LIN {X 0,Y 617.563,Z 761.616,A -85,B 0,C 180,E1 7757.121,E2 7757.121} C_VEL
LIN {X 0,Y 618.923,Z 727.183,A -85,B 0,C 180,E1 7758.711,E2 7758.711} C_VEL
LIN {X 0,Y 620.162,Z 689.828,A -85,B 0,C 180,E1 7759.795,E2 7759.795} C_VEL
LIN {X 0,Y 620.989,Z 629.444,A -85,B 0,C 180,E1 7760.813,E2 7760.813} C_VEL
LIN {X 0,Y 611.333,Z 601.31,A -85,B 0,C 180,E1 7761.822,E2 7761.822} C_VEL
LIN {X 0,Y 611.227,Z 601.31,A -85,B 0,C 180,E1 7766.829,E2 7766.829} C_VEL
LIN {X 0,Y 611.22,Z 601.31,A -85,B 0,C 180,E1 7772.565,E2 7772.565} C_VEL
LIN {X 0,Y 611.08,Z 601.31,A -85,B 0,C 180,E1 7775.407,E2 7775.407} C_VEL
LIN {X 0,Y 607.041,Z 601.31,A -85,B 0,C 180,E1 7777.008,E2 7777.008} C_VEL
LIN {X 0,Y 603.157,Z 601.31,A -85,B 0,C 180,E1 7778.63,E2 7778.63} C_VEL
LIN {X 0,Y 603.164,Z 601.31,A -85,B 0,C 180,E1 7783.244,E2 7783.244} C_VEL
LIN {X 0,Y 603.063,Z 601.31,A -85,B 0,C 180,E1 7789.218,E2 7789.218} C_VEL
LIN {X 0,Y 603.149,Z 601.313,A -85,B 0,C 180,E1 7792.763,E2 7792.763} C_VEL
LIN {X 0,Y 619.848,Z 644.804,A -85,B 0,C 180,E1 7794.111,E2 7794.111} C_VEL
LIN {X 0,Y 624.51,Z 654.896,A -85,B 0,C 180,E1 7794.435,E2 7794.435} C_VEL
LIN {X 0,Y 623.787,Z 712.423,A -85,B 0,C 180,E1 7795.241,E2 7795.241} C_VEL
LIN {X 0,Y 621.771,Z 758.458,A -85,B 0,C 180,E1 7796.44,E2 7796.44} C_VEL
LIN {X 0,Y 619.212,Z 802.863,A -85,B 0,C 180,E1 7798.211,E2 7798.211} C_VEL
LIN {X 0,Y 616.234,Z 843.726,A -85,B 0,C 180,E1 7800.453,E2 7800.453} C_VEL
LIN {X 0,Y 613.148,Z 881.254,A -85,B 0,C 180,E1 7803.152,E2 7803.152} C_VEL
LIN {X 0,Y 610.305,Z 914.42,A -85,B 0,C 180,E1 7806.211,E2 7806.211} C_VEL
LIN {X 0,Y 607.707,Z 941.239,A -85,B 0,C 180,E1 7809.574,E2 7809.574} C_VEL
LIN {X 0,Y 605.902,Z 964.248,A -85,B 0,C 180,E1 7813.291,E2 7813.291} C_VEL
LIN {X 0,Y 604.836,Z 983.335,A -85,B 0,C 180,E1 7817.388,E2 7817.388} C_VEL
LIN {X 0,Y 604.309,Z 996.172,A -85,B 0,C 180,E1 7821.352,E2 7821.352} C_VEL
LIN {X 0,Y 604.218,Z 1003.674,A -85,B 0,C 180,E1 7824.969,E2 7824.969} C_VEL
LIN {X 0,Y 604.188,Z 1007.166,A -85,B 0,C 180,E1 7828.567,E2 7828.567} C_VEL
LIN {X 0,Y 604.173,Z 1006.211,A -85,B 0,C 180,E1 7832.879,E2 7832.879} C_VEL
LIN {X 0,Y 604.211,Z 1001.191,A -85,B 0,C 180,E1 7836.484,E2 7836.484} C_VEL
LIN {X 0,Y 604.502,Z 989.708,A -85,B 0,C 180,E1 7840.84,E2 7840.84} C_VEL
LIN {X 0,Y 605.347,Z 973.833,A -85,B 0,C 180,E1 7844.802,E2 7844.802} C_VEL
LIN {X 0,Y 606.845,Z 952.245,A -85,B 0,C 180,E1 7848.771,E2 7848.771} C_VEL
LIN {X 0,Y 609.432,Z 923.908,A -85,B 0,C 180,E1 7852.71,E2 7852.71} C_VEL
LIN {X 0,Y 612.346,Z 892.188,A -85,B 0,C 180,E1 7855.969,E2 7855.969} C_VEL
LIN {X 0,Y 615.619,Z 855.246,A -85,B 0,C 180,E1 7858.921,E2 7858.921} C_VEL
LIN {X 0,Y 618.871,Z 817.185,A -85,B 0,C 180,E1 7861.277,E2 7861.277} C_VEL
LIN {X 0,Y 622.102,Z 775.086,A -85,B 0,C 180,E1 7863.235,E2 7863.235} C_VEL
LIN {X 0,Y 624.782,Z 729.282,A -85,B 0,C 180,E1 7864.714,E2 7864.714} C_VEL
LIN {X 0,Y 626.356,Z 682.545,A -85,B 0,C 180,E1 7865.608,E2 7865.608} C_VEL
LIN {X 0,Y 626.28,Z 652.86,A -85,B 0,C 180,E1 7866.017,E2 7866.017} C_VEL
LIN {X 0,Y 603.192,Z 601.31,A -85,B 0,C 180,E1 7868.12,E2 7868.12} C_VEL
LIN {X 0,Y 603.121,Z 601.31,A -85,B 0,C 180,E1 7873.245,E2 7873.245} C_VEL
LIN {X 0,Y 603.083,Z 601.31,A -85,B 0,C 180,E1 7879.222,E2 7879.222} C_VEL
LIN {X 0,Y 603.121,Z 601.31,A -85,B 0,C 180,E1 7884.709,E2 7884.709} C_VEL
LIN {X 0,Y 603.248,Z 601.31,A -85,B 0,C 180,E1 7889.85,E2 7889.85} C_VEL
LIN {X 0,Y 603.366,Z 601.31,A -85,B 0,C 180,E1 7894.732,E2 7894.732} C_VEL
LIN {X 0,Y 603.462,Z 601.31,A -85,B 0,C 180,E1 7899.422,E2 7899.422} C_VEL
LIN {X 0,Y 603.517,Z 601.31,A -85,B 0,C 180,E1 7903.97,E2 7903.97} C_VEL
LIN {X 0,Y 603.64,Z 601.31,A -85,B 0,C 180,E1 7909.88,E2 7909.88} C_VEL
LIN {X 0,Y 603.837,Z 601.31,A -85,B 0,C 180,E1 7914.239,E2 7914.239} C_VEL
LIN {X 0,Y 603.903,Z 601.31,A -85,B 0,C 180,E1 7918.561,E2 7918.561} C_VEL
LIN {X 0,Y 603.929,Z 601.31,A -85,B 0,C 180,E1 7922.874,E2 7922.874} C_VEL
LIN {X 0,Y 603.718,Z 601.31,A -85,B 0,C 180,E1 7927.206,E2 7927.206} C_VEL
LIN {X 0,Y 603.614,Z 601.31,A -85,B 0,C 180,E1 7933.052,E2 7933.052} C_VEL
LIN {X 0,Y 603.565,Z 601.31,A -85,B 0,C 180,E1 7937.527,E2 7937.527} C_VEL
LIN {X 0,Y 603.457,Z 601.31,A -85,B 0,C 180,E1 7942.118,E2 7942.118} C_VEL
LIN {X 0,Y 603.371,Z 601.31,A -85,B 0,C 180,E1 7946.865,E2 7946.865} C_VEL
LIN {X 0,Y 603.25,Z 601.31,A -85,B 0,C 180,E1 7951.825,E2 7951.825} C_VEL
LIN {X 0,Y 603.163,Z 601.31,A -85,B 0,C 180,E1 7957.067,E2 7957.067} C_VEL
LIN {X 0,Y 603.143,Z 601.31,A -85,B 0,C 180,E1 7962.696,E2 7962.696} C_VEL
LIN {X 0,Y 603.084,Z 601.31,A -85,B 0,C 180,E1 7967.279,E2 7967.279} C_VEL
LIN {X 0,Y 603.101,Z 601.31,A -85,B 0,C 180,E1 7972.912,E2 7972.912} C_VEL
LIN {X 0,Y 603.252,Z 601.31,A -85,B 0,C 180,E1 7978.624,E2 7978.624} C_VEL
LIN {X 0,Y 603.45,Z 601.31,A -85,B 0,C 180,E1 7981.409,E2 7981.409} C_VEL
LIN {X 0,Y 616.447,Z 643.965,A -85,B 0,C 180,E1 7982.947,E2 7982.947} C_VEL
LIN {X 0,Y 614.768,Z 682.34,A -85,B 0,C 180,E1 7984.248,E2 7984.248} C_VEL
LIN {X 0,Y 612.58,Z 720.776,A -85,B 0,C 180,E1 7986.148,E2 7986.148} C_VEL
LIN {X 0,Y 610.299,Z 754.428,A -85,B 0,C 180,E1 7988.434,E2 7988.434} C_VEL
LIN {X 0,Y 608.249,Z 783.76,A -85,B 0,C 180,E1 7991.1,E2 7991.1} C_VEL
LIN {X 0,Y 606.631,Z 808.095,A -85,B 0,C 180,E1 7994.049,E2 7994.049} C_VEL
LIN {X 0,Y 605.417,Z 828.365,A -85,B 0,C 180,E1 7997.377,E2 7997.377} C_VEL
LIN {X 0,Y 604.627,Z 843.759,A -85,B 0,C 180,E1 8000.985,E2 8000.985} C_VEL
LIN {X 0,Y 604.315,Z 852.718,A -85,B 0,C 180,E1 8004.24,E2 8004.24} C_VEL
LIN {X 0,Y 604.249,Z 857.211,A -85,B 0,C 180,E1 8007.121,E2 8007.121} C_VEL
LIN {X 0,Y 604.192,Z 858.688,A -85,B 0,C 180,E1 8009.996,E2 8009.996} C_VEL
LIN {X 0,Y 604.251,Z 857.119,A -85,B 0,C 180,E1 8012.871,E2 8012.871} C_VEL
LIN {X 0,Y 604.449,Z 850.91,A -85,B 0,C 180,E1 8016.473,E2 8016.473} C_VEL
LIN {X 0,Y 604.799,Z 839.436,A -85,B 0,C 180,E1 8020.096,E2 8020.096} C_VEL
LIN {X 0,Y 605.685,Z 822.808,A -85,B 0,C 180,E1 8023.56,E2 8023.56} C_VEL
LIN {X 0,Y 607.061,Z 802.061,A -85,B 0,C 180,E1 8026.676,E2 8026.676} C_VEL
LIN {X 0,Y 608.764,Z 777.544,A -85,B 0,C 180,E1 8029.441,E2 8029.441} C_VEL
LIN {X 0,Y 610.829,Z 747.106,A -85,B 0,C 180,E1 8032.032,E2 8032.032} C_VEL
LIN {X 0,Y 613.062,Z 712.098,A -85,B 0,C 180,E1 8034.247,E2 8034.247} C_VEL
LIN {X 0,Y 615.193,Z 673.909,A -85,B 0,C 180,E1 8036.001,E2 8036.001} C_VEL
LIN {X 0,Y 615.776,Z 640.775,A -85,B 0,C 180,E1 8037.082,E2 8037.082} C_VEL
LIN {X 0,Y 603.379,Z 601.31,A -85,B 0,C 180,E1 8038.514,E2 8038.514} C_VEL
LIN {X 0,Y 603.18,Z 601.31,A -85,B 0,C 180,E1 8044.028,E2 8044.028} C_VEL
LIN {X 0,Y 603.145,Z 601.31,A -85,B 0,C 180,E1 8048.901,E2 8048.901} C_VEL
LIN {X 0,Y 603.167,Z 601.31,A -85,B 0,C 180,E1 8054.693,E2 8054.693} C_VEL
LIN {X 0,Y 603.069,Z 601.31,A -85,B 0,C 180,E1 8059.226,E2 8059.226} C_VEL
LIN {X 0,Y 603.126,Z 601.31,A -85,B 0,C 180,E1 8064.714,E2 8064.714} C_VEL
LIN {X 0,Y 603.244,Z 601.31,A -85,B 0,C 180,E1 8069.853,E2 8069.853} C_VEL
LIN {X 0,Y 603.393,Z 601.31,A -85,B 0,C 180,E1 8074.737,E2 8074.737} C_VEL
LIN {X 0,Y 603.41,Z 601.31,A -85,B 0,C 180,E1 8078.339,E2 8078.339} C_VEL
LIN {X 0,Y 613.169,Z 634.007,A -85,B 0,C 180,E1 8079.179,E2 8079.179} C_VEL
LIN {X 0,Y 612.014,Z 695.654,A -85,B 0,C 180,E1 8080.132,E2 8080.132} C_VEL
LIN {X 0,Y 610.916,Z 730.893,A -85,B 0,C 180,E1 8081.243,E2 8081.243} C_VEL
LIN {X 0,Y 609.315,Z 764.343,A -85,B 0,C 180,E1 8082.898,E2 8082.898} C_VEL
LIN {X 0,Y 607.883,Z 793.927,A -85,B 0,C 180,E1 8085.018,E2 8085.018} C_VEL
LIN {X 0,Y 606.55,Z 819.418,A -85,B 0,C 180,E1 8087.562,E2 8087.562} C_VEL
LIN {X 0,Y 605.622,Z 840.01,A -85,B 0,C 180,E1 8090.463,E2 8090.463} C_VEL
LIN {X 0,Y 605.138,Z 854.695,A -85,B 0,C 180,E1 8093.534,E2 8093.534} C_VEL
LIN {X 0,Y 604.907,Z 863.079,A -85,B 0,C 180,E1 8096.412,E2 8096.412} C_VEL
LIN {X 0,Y 604.827,Z 866.274,A -85,B 0,C 180,E1 8098.567,E2 8098.567} C_VEL
LIN {X 0,Y 604.876,Z 866.684,A -85,B 0,C 180,E1 8101.437,E2 8101.437} C_VEL
LIN {X 0,Y 605.13,Z 862.587,A -85,B 0,C 180,E1 8104.309,E2 8104.309} C_VEL
LIN {X 0,Y 605.545,Z 853.627,A -85,B 0,C 180,E1 8107.187,E2 8107.187} C_VEL
LIN {X 0,Y 606.305,Z 837.945,A -85,B 0,C 180,E1 8110.256,E2 8110.256} C_VEL
LIN {X 0,Y 607.271,Z 817.336,A -85,B 0,C 180,E1 8112.976,E2 8112.976} C_VEL
LIN {X 0,Y 608.696,Z 792.26,A -85,B 0,C 180,E1 8115.335,E2 8115.335} C_VEL
LIN {X 0,Y 610.075,Z 762.601,A -85,B 0,C 180,E1 8117.338,E2 8117.338} C_VEL
LIN {X 0,Y 611.517,Z 728.166,A -85,B 0,C 180,E1 8118.95,E2 8118.95} C_VEL
LIN {X 0,Y 612.94,Z 689.262,A -85,B 0,C 180,E1 8120.098,E2 8120.098} C_VEL
LIN {X 0,Y 613.832,Z 631.246,A -85,B 0,C 180,E1 8121.105,E2 8121.105} C_VEL
LIN {X 0,Y 603.386,Z 601.31,A -85,B 0,C 180,E1 8122.222,E2 8122.222} C_VEL
LIN {X 0,Y 603.346,Z 601.31,A -85,B 0,C 180,E1 8126.87,E2 8126.87} C_VEL
LIN {X 0,Y 603.271,Z 601.31,A -85,B 0,C 180,E1 8131.828,E2 8131.828} C_VEL
LIN {X 0,Y 603.187,Z 601.31,A -85,B 0,C 180,E1 8137.069,E2 8137.069} C_VEL
LIN {X 0,Y 603.157,Z 601.31,A -85,B 0,C 180,E1 8138.63,E2 8138.63} C_VEL
LIN {X 0,Y 600.687,Z 601.31,A -85,B 0,C 180,E1 8139.854,E2 8139.854} C_VEL
LIN {X 0,Y 595.291,Z 601.31,A -85,B 0,C 180,E1 8141.684,E2 8141.684} C_VEL
LIN {X 0,Y 595.198,Z 601.31,A -85,B 0,C 180,E1 8141.896,E2 8141.896} C_VEL
LIN {X 0,Y 595.189,Z 601.31,A -85,B 0,C 180,E1 8146.585,E2 8146.585} C_VEL
LIN {X 0,Y 595.209,Z 601.31,A -85,B 0,C 180,E1 8152.319,E2 8152.319} C_VEL
LIN {X 0,Y 613.922,Z 649.623,A -85,B 0,C 180,E1 8153.902,E2 8153.902} C_VEL
LIN {X 0,Y 617.375,Z 657.627,A -85,B 0,C 180,E1 8154.155,E2 8154.155} C_VEL
LIN {X 0,Y 616.536,Z 713.468,A -85,B 0,C 180,E1 8154.963,E2 8154.963} C_VEL
LIN {X 0,Y 614.403,Z 759.623,A -85,B 0,C 180,E1 8156.196,E2 8156.196} C_VEL
LIN {X 0,Y 611.618,Z 805.625,A -85,B 0,C 180,E1 8158.08,E2 8158.08} C_VEL
LIN {X 0,Y 608.303,Z 848.784,A -85,B 0,C 180,E1 8160.546,E2 8160.546} C_VEL
LIN {X 0,Y 604.87,Z 888.615,A -85,B 0,C 180,E1 8163.582,E2 8163.582} C_VEL
LIN {X 0,Y 601.741,Z 923.451,A -85,B 0,C 180,E1 8167.063,E2 8167.063} C_VEL
LIN {X 0,Y 599.678,Z 946.379,A -85,B 0,C 180,E1 8170.06,E2 8170.06} C_VEL
LIN {X 0,Y 597.852,Z 969.915,A -85,B 0,C 180,E1 8174.161,E2 8174.161} C_VEL
LIN {X 0,Y 596.736,Z 988.527,A -85,B 0,C 180,E1 8178.655,E2 8178.655} C_VEL
LIN {X 0,Y 596.284,Z 999.644,A -85,B 0,C 180,E1 8182.705,E2 8182.705} C_VEL
LIN {X 0,Y 596.209,Z 1004.651,A -85,B 0,C 180,E1 8185.631,E2 8185.631} C_VEL
LIN {X 0,Y 596.225,Z 1007.5,A -85,B 0,C 180,E1 8190.004,E2 8190.004} C_VEL
LIN {X 0,Y 596.215,Z 1004.643,A -85,B 0,C 180,E1 8194.377,E2 8194.377} C_VEL
LIN {X 0,Y 596.356,Z 997.729,A -85,B 0,C 180,E1 8198.17,E2 8198.17} C_VEL
LIN {X 0,Y 596.971,Z 984.297,A -85,B 0,C 180,E1 8202.516,E2 8202.516} C_VEL
LIN {X 0,Y 598.066,Z 966.147,A -85,B 0,C 180,E1 8206.564,E2 8206.564} C_VEL
LIN {X 0,Y 599.991,Z 942.505,A -85,B 0,C 180,E1 8210.516,E2 8210.516} C_VEL
LIN {X 0,Y 602.738,Z 913.178,A -85,B 0,C 180,E1 8214.115,E2 8214.115} C_VEL
LIN {X 0,Y 606.18,Z 876.8,A -85,B 0,C 180,E1 8217.546,E2 8217.546} C_VEL
LIN {X 0,Y 609.936,Z 836.375,A -85,B 0,C 180,E1 8220.465,E2 8220.465} C_VEL
LIN {X 0,Y 613.729,Z 792.251,A -85,B 0,C 180,E1 8222.838,E2 8222.838} C_VEL
LIN {X 0,Y 616.821,Z 747.376,A -85,B 0,C 180,E1 8224.549,E2 8224.549} C_VEL
LIN {X 0,Y 618.891,Z 702.958,A -85,B 0,C 180,E1 8225.646,E2 8225.646} C_VEL
LIN {X 0,Y 619.293,Z 655.089,A -85,B 0,C 180,E1 8226.364,E2 8226.364} C_VEL
LIN {X 0,Y 595.27,Z 601.31,A -85,B 0,C 180,E1 8228.572,E2 8228.572} C_VEL
LIN {X 0,Y 595.226,Z 601.31,A -85,B 0,C 180,E1 8234.549,E2 8234.549} C_VEL
LIN {X 0,Y 595.124,Z 601.31,A -85,B 0,C 180,E1 8240.476,E2 8240.476} C_VEL
LIN {X 0,Y 595.218,Z 601.31,A -85,B 0,C 180,E1 8245.948,E2 8245.948} C_VEL
LIN {X 0,Y 595.351,Z 601.31,A -85,B 0,C 180,E1 8251.086,E2 8251.086} C_VEL
LIN {X 0,Y 595.52,Z 601.31,A -85,B 0,C 180,E1 8256.353,E2 8256.353} C_VEL
LIN {X 0,Y 595.578,Z 601.31,A -85,B 0,C 180,E1 8262.226,E2 8262.226} C_VEL
LIN {X 0,Y 595.721,Z 601.31,A -85,B 0,C 180,E1 8268.26,E2 8268.26} C_VEL
LIN {X 0,Y 595.925,Z 601.31,A -85,B 0,C 180,E1 8274.162,E2 8274.162} C_VEL
LIN {X 0,Y 596.002,Z 601.31,A -85,B 0,C 180,E1 8278.542,E2 8278.542} C_VEL
LIN {X 0,Y 596.025,Z 601.31,A -85,B 0,C 180,E1 8282.912,E2 8282.912} C_VEL
LIN {X 0,Y 595.825,Z 601.31,A -85,B 0,C 180,E1 8287.318,E2 8287.318} C_VEL
LIN {X 0,Y 595.77,Z 601.31,A -85,B 0,C 180,E1 8291.735,E2 8291.735} C_VEL
LIN {X 0,Y 595.652,Z 601.31,A -85,B 0,C 180,E1 8296.244,E2 8296.244} C_VEL
LIN {X 0,Y 595.568,Z 601.31,A -85,B 0,C 180,E1 8300.859,E2 8300.859} C_VEL
LIN {X 0,Y 595.449,Z 601.31,A -85,B 0,C 180,E1 8305.624,E2 8305.624} C_VEL
LIN {X 0,Y 595.331,Z 601.31,A -85,B 0,C 180,E1 8310.59,E2 8310.59} C_VEL
LIN {X 0,Y 595.254,Z 601.31,A -85,B 0,C 180,E1 8315.824,E2 8315.824} C_VEL
LIN {X 0,Y 595.202,Z 601.31,A -85,B 0,C 180,E1 8321.43,E2 8321.43} C_VEL
LIN {X 0,Y 595.21,Z 601.31,A -85,B 0,C 180,E1 8326.575,E2 8326.575} C_VEL
LIN {X 0,Y 595.138,Z 601.31,A -85,B 0,C 180,E1 8332.331,E2 8332.331} C_VEL
LIN {X 0,Y 595.261,Z 601.31,A -85,B 0,C 180,E1 8337.682,E2 8337.682} C_VEL
LIN {X 0,Y 595.462,Z 601.31,A -85,B 0,C 180,E1 8341.009,E2 8341.009} C_VEL
LIN {X 0,Y 609.257,Z 645.924,A -85,B 0,C 180,E1 8342.681,E2 8342.681} C_VEL
LIN {X 0,Y 607.339,Z 684.919,A -85,B 0,C 180,E1 8344.041,E2 8344.041} C_VEL
LIN {X 0,Y 605.028,Z 722.818,A -85,B 0,C 180,E1 8345.988,E2 8345.988} C_VEL
LIN {X 0,Y 602.561,Z 756.799,A -85,B 0,C 180,E1 8348.38,E2 8348.38} C_VEL
LIN {X 0,Y 600.512,Z 785.619,A -85,B 0,C 180,E1 8351.058,E2 8351.058} C_VEL
LIN {X 0,Y 598.811,Z 810.529,A -85,B 0,C 180,E1 8354.139,E2 8354.139} C_VEL
LIN {X 0,Y 597.536,Z 831.1,A -85,B 0,C 180,E1 8357.625,E2 8357.625} C_VEL
LIN {X 0,Y 596.823,Z 845.826,A -85,B 0,C 180,E1 8361.234,E2 8361.234} C_VEL
LIN {X 0,Y 596.552,Z 855.105,A -85,B 0,C 180,E1 8364.896,E2 8364.896} C_VEL
LIN {X 0,Y 596.316,Z 859.334,A -85,B 0,C 180,E1 8368.54,E2 8368.54} C_VEL
LIN {X 0,Y 596.408,Z 859.266,A -85,B 0,C 180,E1 8371.452,E2 8371.452} C_VEL
LIN {X 0,Y 596.578,Z 854.94,A -85,B 0,C 180,E1 8375.096,E2 8375.096} C_VEL
LIN {X 0,Y 596.815,Z 845.545,A -85,B 0,C 180,E1 8378.758,E2 8378.758} C_VEL
LIN {X 0,Y 597.572,Z 830.585,A -85,B 0,C 180,E1 8382.384,E2 8382.384} C_VEL
LIN {X 0,Y 598.715,Z 811.193,A -85,B 0,C 180,E1 8385.678,E2 8385.678} C_VEL
LIN {X 0,Y 600.359,Z 787.619,A -85,B 0,C 180,E1 8388.639,E2 8388.639} C_VEL
LIN {X 0,Y 602.469,Z 758.418,A -85,B 0,C 180,E1 8391.398,E2 8391.398} C_VEL
LIN {X 0,Y 604.898,Z 724.609,A -85,B 0,C 180,E1 8393.809,E2 8393.809} C_VEL
LIN {X 0,Y 607.316,Z 686.329,A -85,B 0,C 180,E1 8395.808,E2 8395.808} C_VEL
LIN {X 0,Y 609.194,Z 647.276,A -85,B 0,C 180,E1 8397.192,E2 8397.192} C_VEL
LIN {X 0,Y 597.28,Z 607.328,A -85,B 0,C 180,E1 8398.691,E2 8398.691} C_VEL
LIN {X 0,Y 595.418,Z 601.31,A -85,B 0,C 180,E1 8398.91,E2 8398.91} C_VEL
LIN {X 0,Y 595.293,Z 601.31,A -85,B 0,C 180,E1 8404.049,E2 8404.049} C_VEL
LIN {X 0,Y 595.174,Z 601.31,A -85,B 0,C 180,E1 8410.222,E2 8410.222} C_VEL
LIN {X 0,Y 595.248,Z 601.31,A -85,B 0,C 180,E1 8415.453,E2 8415.453} C_VEL
LIN {X 0,Y 595.126,Z 601.31,A -85,B 0,C 180,E1 8420.481,E2 8420.481} C_VEL
LIN {X 0,Y 595.227,Z 601.31,A -85,B 0,C 180,E1 8425.953,E2 8425.953} C_VEL
LIN {X 0,Y 595.349,Z 601.31,A -85,B 0,C 180,E1 8431.09,E2 8431.09} C_VEL
LIN {X 0,Y 595.511,Z 601.31,A -85,B 0,C 180,E1 8436.335,E2 8436.335} C_VEL
LIN {X 0,Y 595.505,Z 601.31,A -85,B 0,C 180,E1 8438.036,E2 8438.036} C_VEL
LIN {X 0,Y 605.742,Z 636.116,A -85,B 0,C 180,E1 8438.948,E2 8438.948} C_VEL
LIN {X 0,Y 604.561,Z 696.009,A -85,B 0,C 180,E1 8439.893,E2 8439.893} C_VEL
LIN {X 0,Y 603.363,Z 731.904,A -85,B 0,C 180,E1 8441.047,E2 8441.047} C_VEL
LIN {X 0,Y 601.721,Z 764.904,A -85,B 0,C 180,E1 8442.703,E2 8442.703} C_VEL
LIN {X 0,Y 600.188,Z 794.251,A -85,B 0,C 180,E1 8444.821,E2 8444.821} C_VEL
LIN {X 0,Y 598.823,Z 819.942,A -85,B 0,C 180,E1 8447.399,E2 8447.399} C_VEL
LIN {X 0,Y 597.858,Z 840.706,A -85,B 0,C 180,E1 8450.338,E2 8450.338} C_VEL
LIN {X 0,Y 597.332,Z 855.512,A -85,B 0,C 180,E1 8453.449,E2 8453.449} C_VEL
LIN {X 0,Y 597.074,Z 864.018,A -85,B 0,C 180,E1 8456.365,E2 8456.365} C_VEL
LIN {X 0,Y 597.006,Z 867.283,A -85,B 0,C 180,E1 8458.548,E2 8458.548} C_VEL
LIN {X 0,Y 597.055,Z 867.756,A -85,B 0,C 180,E1 8461.456,E2 8461.456} C_VEL
LIN {X 0,Y 597.349,Z 863.684,A -85,B 0,C 180,E1 8464.365,E2 8464.365} C_VEL
LIN {X 0,Y 597.793,Z 854.722,A -85,B 0,C 180,E1 8467.281,E2 8467.281} C_VEL
LIN {X 0,Y 598.529,Z 840.139,A -85,B 0,C 180,E1 8470.207,E2 8470.207} C_VEL
LIN {X 0,Y 599.587,Z 820.021,A -85,B 0,C 180,E1 8472.96,E2 8472.96} C_VEL
LIN {X 0,Y 601.09,Z 794.425,A -85,B 0,C 180,E1 8475.44,E2 8475.44} C_VEL
LIN {X 0,Y 602.552,Z 765.2,A -85,B 0,C 180,E1 8477.465,E2 8477.465} C_VEL
LIN {X 0,Y 604.132,Z 730.304,A -85,B 0,C 180,E1 8479.159,E2 8479.159} C_VEL
LIN {X 0,Y 605.615,Z 691.724,A -85,B 0,C 180,E1 8480.346,E2 8480.346} C_VEL
LIN {X 0,Y 606.712,Z 632.927,A -85,B 0,C 180,E1 8481.41,E2 8481.41} C_VEL
LIN {X 0,Y 595.466,Z 601.31,A -85,B 0,C 180,E1 8482.663,E2 8482.663} C_VEL
LIN {X 0,Y 595.399,Z 601.31,A -85,B 0,C 180,E1 8487.259,E2 8487.259} C_VEL
LIN {X 0,Y 595.27,Z 601.31,A -85,B 0,C 180,E1 8492.869,E2 8492.869} C_VEL
LIN {X 0,Y 595.216,Z 601.31,A -85,B 0,C 180,E1 8497.901,E2 8497.901} C_VEL
LIN {X 0,Y 595.198,Z 601.31,A -85,B 0,C 180,E1 8501.896,E2 8501.896} C_VEL
LIN {X 0,Y 593.944,Z 601.31,A -85,B 0,C 180,E1 8502.731,E2 8502.731} C_VEL
LIN {X 0,Y 587.363,Z 601.31,A -85,B 0,C 180,E1 8505.003,E2 8505.003} C_VEL
LIN {X 0,Y 587.275,Z 601.31,A -85,B 0,C 180,E1 8505.218,E2 8505.218} C_VEL
LIN {X 0,Y 587.191,Z 601.31,A -85,B 0,C 180,E1 8510.714,E2 8510.714} C_VEL
LIN {X 0,Y 587.241,Z 601.31,A -85,B 0,C 180,E1 8511.862,E2 8511.862} C_VEL
LIN {X 0,Y 607.768,Z 653.878,A -85,B 0,C 180,E1 8513.664,E2 8513.664} C_VEL
LIN {X 0,Y 610.278,Z 659.489,A -85,B 0,C 180,E1 8513.852,E2 8513.852} C_VEL
LIN {X 0,Y 609.403,Z 712.874,A -85,B 0,C 180,E1 8514.638,E2 8514.638} C_VEL
LIN {X 0,Y 607.174,Z 759.213,A -85,B 0,C 180,E1 8515.889,E2 8515.889} C_VEL
LIN {X 0,Y 604.257,Z 804.885,A -85,B 0,C 180,E1 8517.779,E2 8517.779} C_VEL
LIN {X 0,Y 600.75,Z 848.405,A -85,B 0,C 180,E1 8520.289,E2 8520.289} C_VEL
LIN {X 0,Y 597.259,Z 887.99,A -85,B 0,C 180,E1 8523.343,E2 8523.343} C_VEL
LIN {X 0,Y 594.021,Z 922.55,A -85,B 0,C 180,E1 8526.833,E2 8526.833} C_VEL
LIN {X 0,Y 591.617,Z 950.852,A -85,B 0,C 180,E1 8530.557,E2 8530.557} C_VEL
LIN {X 0,Y 590.003,Z 970.896,A -85,B 0,C 180,E1 8534.158,E2 8534.158} C_VEL
LIN {X 0,Y 588.887,Z 988.526,A -85,B 0,C 180,E1 8538.502,E2 8538.502} C_VEL
LIN {X 0,Y 588.398,Z 999.644,A -85,B 0,C 180,E1 8542.606,E2 8542.606} C_VEL
LIN {X 0,Y 588.316,Z 1004.651,A -85,B 0,C 180,E1 8545.573,E2 8545.573} C_VEL
LIN {X 0,Y 588.339,Z 1007.5,A -85,B 0,C 180,E1 8550.004,E2 8550.004} C_VEL
LIN {X 0,Y 588.323,Z 1004.642,A -85,B 0,C 180,E1 8554.435,E2 8554.435} C_VEL
LIN {X 0,Y 588.475,Z 997.466,A -85,B 0,C 180,E1 8558.382,E2 8558.382} C_VEL
LIN {X 0,Y 589.133,Z 984.099,A -85,B 0,C 180,E1 8562.741,E2 8562.741} C_VEL
LIN {X 0,Y 590.259,Z 966.146,A -85,B 0,C 180,E1 8566.79,E2 8566.79} C_VEL
LIN {X 0,Y 592.021,Z 945.709,A -85,B 0,C 180,E1 8570.218,E2 8570.218} C_VEL
LIN {X 0,Y 594.687,Z 917.089,A -85,B 0,C 180,E1 8573.865,E2 8573.865} C_VEL
LIN {X 0,Y 597.911,Z 884.321,A -85,B 0,C 180,E1 8577.143,E2 8577.143} C_VEL
LIN {X 0,Y 601.521,Z 847.907,A -85,B 0,C 180,E1 8579.998,E2 8579.998} C_VEL
LIN {X 0,Y 605.428,Z 805.564,A -85,B 0,C 180,E1 8582.525,E2 8582.525} C_VEL
LIN {X 0,Y 608.957,Z 760.192,A -85,B 0,C 180,E1 8584.481,E2 8584.481} C_VEL
LIN {X 0,Y 611.671,Z 712.284,A -85,B 0,C 180,E1 8585.835,E2 8585.835} C_VEL
LIN {X 0,Y 612.724,Z 658.182,A -85,B 0,C 180,E1 8586.686,E2 8586.686} C_VEL
LIN {X 0,Y 587.29,Z 601.31,A -85,B 0,C 180,E1 8589.059,E2 8589.059} C_VEL
LIN {X 0,Y 587.299,Z 601.31,A -85,B 0,C 180,E1 8594.16,E2 8594.16} C_VEL
LIN {X 0,Y 587.249,Z 601.31,A -85,B 0,C 180,E1 8599.839,E2 8599.839} C_VEL
LIN {X 0,Y 587.291,Z 601.31,A -85,B 0,C 180,E1 8605.656,E2 8605.656} C_VEL
LIN {X 0,Y 587.449,Z 601.31,A -85,B 0,C 180,E1 8611.286,E2 8611.286} C_VEL
LIN {X 0,Y 587.533,Z 601.31,A -85,B 0,C 180,E1 8615.633,E2 8615.633} C_VEL
LIN {X 0,Y 587.67,Z 601.31,A -85,B 0,C 180,E1 8620.419,E2 8620.419} C_VEL
LIN {X 0,Y 587.714,Z 601.31,A -85,B 0,C 180,E1 8625.061,E2 8625.061} C_VEL
LIN {X 0,Y 587.829,Z 601.31,A -85,B 0,C 180,E1 8629.605,E2 8629.605} C_VEL
LIN {X 0,Y 588.02,Z 601.31,A -85,B 0,C 180,E1 8634.083,E2 8634.083} C_VEL
LIN {X 0,Y 588.119,Z 601.31,A -85,B 0,C 180,E1 8638.522,E2 8638.522} C_VEL
LIN {X 0,Y 588.121,Z 601.31,A -85,B 0,C 180,E1 8642.951,E2 8642.951} C_VEL
LIN {X 0,Y 587.943,Z 601.31,A -85,B 0,C 180,E1 8647.4,E2 8647.4} C_VEL
LIN {X 0,Y 587.848,Z 601.31,A -85,B 0,C 180,E1 8651.895,E2 8651.895} C_VEL
LIN {X 0,Y 587.711,Z 601.31,A -85,B 0,C 180,E1 8657.449,E2 8657.449} C_VEL
LIN {X 0,Y 587.597,Z 601.31,A -85,B 0,C 180,E1 8662.748,E2 8662.748} C_VEL
LIN {X 0,Y 587.46,Z 601.31,A -85,B 0,C 180,E1 8667.654,E2 8667.654} C_VEL
LIN {X 0,Y 587.373,Z 601.31,A -85,B 0,C 180,E1 8672.791,E2 8672.791} C_VEL
LIN {X 0,Y 587.245,Z 601.31,A -85,B 0,C 180,E1 8678.249,E2 8678.249} C_VEL
LIN {X 0,Y 587.367,Z 601.31,A -85,B 0,C 180,E1 8684.133,E2 8684.133} C_VEL
LIN {X 0,Y 587.249,Z 601.31,A -85,B 0,C 180,E1 8689.826,E2 8689.826} C_VEL
LIN {X 0,Y 587.303,Z 601.31,A -85,B 0,C 180,E1 8695.626,E2 8695.626} C_VEL
LIN {X 0,Y 587.541,Z 601.31,A -85,B 0,C 180,E1 8700.584,E2 8700.584} C_VEL
LIN {X 0,Y 602.055,Z 645.753,A -85,B 0,C 180,E1 8702.335,E2 8702.335} C_VEL
LIN {X 0,Y 600.184,Z 685.101,A -85,B 0,C 180,E1 8703.721,E2 8703.721} C_VEL
LIN {X 0,Y 597.8,Z 722.487,A -85,B 0,C 180,E1 8705.65,E2 8705.65} C_VEL
LIN {X 0,Y 595.125,Z 756.62,A -85,B 0,C 180,E1 8708.076,E2 8708.076} C_VEL
LIN {X 0,Y 592.85,Z 786.216,A -85,B 0,C 180,E1 8710.876,E2 8710.876} C_VEL
LIN {X 0,Y 591.114,Z 810.794,A -85,B 0,C 180,E1 8713.927,E2 8713.927} C_VEL
LIN {X 0,Y 589.815,Z 831.412,A -85,B 0,C 180,E1 8717.411,E2 8717.411} C_VEL
LIN {X 0,Y 589.005,Z 846.618,A -85,B 0,C 180,E1 8721.117,E2 8721.117} C_VEL
LIN {X 0,Y 588.72,Z 856.021,A -85,B 0,C 180,E1 8724.828,E2 8724.828} C_VEL
LIN {X 0,Y 588.479,Z 860.315,A -85,B 0,C 180,E1 8728.521,E2 8728.521} C_VEL
LIN {X 0,Y 588.594,Z 860.244,A -85,B 0,C 180,E1 8731.471,E2 8731.471} C_VEL
LIN {X 0,Y 588.746,Z 855.856,A -85,B 0,C 180,E1 8735.164,E2 8735.164} C_VEL
LIN {X 0,Y 588.999,Z 846.334,A -85,B 0,C 180,E1 8738.875,E2 8738.875} C_VEL
LIN {X 0,Y 589.829,Z 830.909,A -85,B 0,C 180,E1 8742.595,E2 8742.595} C_VEL
LIN {X 0,Y 591.04,Z 811.217,A -85,B 0,C 180,E1 8745.923,E2 8745.923} C_VEL
LIN {X 0,Y 592.84,Z 786.384,A -85,B 0,C 180,E1 8749.016,E2 8749.016} C_VEL
LIN {X 0,Y 595.265,Z 755.377,A -85,B 0,C 180,E1 8751.937,E2 8751.937} C_VEL
LIN {X 0,Y 597.919,Z 721.039,A -85,B 0,C 180,E1 8754.343,E2 8754.343} C_VEL
LIN {X 0,Y 600.227,Z 684.893,A -85,B 0,C 180,E1 8756.196,E2 8756.196} C_VEL
LIN {X 0,Y 601.662,Z 645.593,A -85,B 0,C 180,E1 8757.598,E2 8757.598} C_VEL
LIN {X 0,Y 588.754,Z 605.604,A -85,B 0,C 180,E1 8759.166,E2 8759.166} C_VEL
LIN {X 0,Y 587.482,Z 601.31,A -85,B 0,C 180,E1 8759.338,E2 8759.338} C_VEL
LIN {X 0,Y 587.358,Z 601.31,A -85,B 0,C 180,E1 8764.573,E2 8764.573} C_VEL
LIN {X 0,Y 587.277,Z 601.31,A -85,B 0,C 180,E1 8770.161,E2 8770.161} C_VEL
LIN {X 0,Y 587.33,Z 601.31,A -85,B 0,C 180,E1 8775.864,E2 8775.864} C_VEL
LIN {X 0,Y 587.223,Z 601.31,A -85,B 0,C 180,E1 8781.749,E2 8781.749} C_VEL
LIN {X 0,Y 587.342,Z 601.31,A -85,B 0,C 180,E1 8787.207,E2 8787.207} C_VEL
LIN {X 0,Y 587.487,Z 601.31,A -85,B 0,C 180,E1 8792.347,E2 8792.347} C_VEL
LIN {X 0,Y 587.581,Z 601.31,A -85,B 0,C 180,E1 8797.7,E2 8797.7} C_VEL
LIN {X 0,Y 598.348,Z 637.12,A -85,B 0,C 180,E1 8798.691,E2 8798.691} C_VEL
LIN {X 0,Y 597.117,Z 696.435,A -85,B 0,C 180,E1 8799.649,E2 8799.649} C_VEL
LIN {X 0,Y 595.853,Z 731.823,A -85,B 0,C 180,E1 8800.799,E2 8800.799} C_VEL
LIN {X 0,Y 594.135,Z 765.523,A -85,B 0,C 180,E1 8802.507,E2 8802.507} C_VEL
LIN {X 0,Y 592.488,Z 795.647,A -85,B 0,C 180,E1 8804.714,E2 8804.714} C_VEL
LIN {X 0,Y 591.091,Z 820.616,A -85,B 0,C 180,E1 8807.253,E2 8807.253} C_VEL
LIN {X 0,Y 590.073,Z 841.362,A -85,B 0,C 180,E1 8810.209,E2 8810.209} C_VEL
LIN {X 0,Y 589.536,Z 856.324,A -85,B 0,C 180,E1 8813.362,E2 8813.362} C_VEL
LIN {X 0,Y 589.251,Z 864.948,A -85,B 0,C 180,E1 8816.317,E2 8816.317} C_VEL
LIN {X 0,Y 589.194,Z 868.284,A -85,B 0,C 180,E1 8818.529,E2 8818.529} C_VEL
LIN {X 0,Y 589.236,Z 868.824,A -85,B 0,C 180,E1 8821.475,E2 8821.475} C_VEL
LIN {X 0,Y 589.575,Z 864.786,A -85,B 0,C 180,E1 8824.423,E2 8824.423} C_VEL
LIN {X 0,Y 590.028,Z 855.866,A -85,B 0,C 180,E1 8827.377,E2 8827.377} C_VEL
LIN {X 0,Y 590.843,Z 841.246,A -85,B 0,C 180,E1 8830.341,E2 8830.341} C_VEL
LIN {X 0,Y 591.952,Z 821.126,A -85,B 0,C 180,E1 8833.13,E2 8833.13} C_VEL
LIN {X 0,Y 593.479,Z 796.558,A -85,B 0,C 180,E1 8835.548,E2 8835.548} C_VEL
LIN {X 0,Y 595.065,Z 766.964,A -85,B 0,C 180,E1 8837.655,E2 8837.655} C_VEL
LIN {X 0,Y 596.736,Z 733.152,A -85,B 0,C 180,E1 8839.345,E2 8839.345} C_VEL
LIN {X 0,Y 598.364,Z 694.39,A -85,B 0,C 180,E1 8840.6,E2 8840.6} C_VEL
LIN {X 0,Y 599.829,Z 635.292,A -85,B 0,C 180,E1 8841.707,E2 8841.707} C_VEL
LIN {X 0,Y 587.538,Z 601.31,A -85,B 0,C 180,E1 8843.171,E2 8843.171} C_VEL
LIN {X 0,Y 587.466,Z 601.31,A -85,B 0,C 180,E1 8848.734,E2 8848.734} C_VEL
LIN {X 0,Y 587.371,Z 601.31,A -85,B 0,C 180,E1 8854.571,E2 8854.571} C_VEL
LIN {X 0,Y 587.308,Z 601.31,A -85,B 0,C 180,E1 8860.156,E2 8860.156} C_VEL
LIN {X 0,Y 587.275,Z 601.31,A -85,B 0,C 180,E1 8865.218,E2 8865.218} C_VEL
LIN {X 0,Y 584.706,Z 601.31,A -85,B 0,C 180,E1 8866.476,E2 8866.476} C_VEL
LIN {X 0,Y 579.298,Z 601.31,A -85,B 0,C 180,E1 8868.358,E2 8868.358} C_VEL
LIN {X 0,Y 579.217,Z 601.31,A -85,B 0,C 180,E1 8868.576,E2 8868.576} C_VEL
LIN {X 0,Y 579.331,Z 601.31,A -85,B 0,C 180,E1 8871.368,E2 8871.368} C_VEL
LIN {X 0,Y 594.273,Z 640.75,A -85,B 0,C 180,E1 8872.81,E2 8872.81} C_VEL
LIN {X 0,Y 603.184,Z 663.029,A -85,B 0,C 180,E1 8873.555,E2 8873.555} C_VEL
LIN {X 0,Y 602.257,Z 713.576,A -85,B 0,C 180,E1 8874.328,E2 8874.328} C_VEL
LIN {X 0,Y 599.925,Z 759.226,A -85,B 0,C 180,E1 8875.584,E2 8875.584} C_VEL
LIN {X 0,Y 596.858,Z 804.902,A -85,B 0,C 180,E1 8877.505,E2 8877.505} C_VEL
LIN {X 0,Y 593.288,Z 847.783,A -85,B 0,C 180,E1 8880.011,E2 8880.011} C_VEL
LIN {X 0,Y 589.659,Z 887.119,A -85,B 0,C 180,E1 8883.075,E2 8883.075} C_VEL
LIN {X 0,Y 586.337,Z 921.481,A -85,B 0,C 180,E1 8886.578,E2 8886.578} C_VEL
LIN {X 0,Y 583.836,Z 949.473,A -85,B 0,C 180,E1 8890.287,E2 8890.287} C_VEL
LIN {X 0,Y 582.21,Z 970.763,A -85,B 0,C 180,E1 8893.937,E2 8893.937} C_VEL
LIN {X 0,Y 581.034,Z 988.526,A -85,B 0,C 180,E1 8898.344,E2 8898.344} C_VEL
LIN {X 0,Y 580.501,Z 999.853,A -85,B 0,C 180,E1 8902.606,E2 8902.606} C_VEL
LIN {X 0,Y 580.422,Z 1004.65,A -85,B 0,C 180,E1 8905.512,E2 8905.512} C_VEL
LIN {X 0,Y 580.439,Z 1007.5,A -85,B 0,C 180,E1 8910.004,E2 8910.004} C_VEL
LIN {X 0,Y 580.43,Z 1004.642,A -85,B 0,C 180,E1 8914.496,E2 8914.496} C_VEL
LIN {X 0,Y 580.562,Z 998.06,A -85,B 0,C 180,E1 8918.257,E2 8918.257} C_VEL
LIN {X 0,Y 581.263,Z 984.485,A -85,B 0,C 180,E1 8922.806,E2 8922.806} C_VEL
LIN {X 0,Y 582.384,Z 967.809,A -85,B 0,C 180,E1 8926.634,E2 8926.634} C_VEL
LIN {X 0,Y 584.383,Z 942.873,A -85,B 0,C 180,E1 8930.76,E2 8930.76} C_VEL
LIN {X 0,Y 587.532,Z 911.288,A -85,B 0,C 180,E1 8934.721,E2 8934.721} C_VEL
LIN {X 0,Y 591.269,Z 875.962,A -85,B 0,C 180,E1 8938.132,E2 8938.132} C_VEL
LIN {X 0,Y 595.448,Z 835.629,A -85,B 0,C 180,E1 8941.115,E2 8941.115} C_VEL
LIN {X 0,Y 599.471,Z 792.555,A -85,B 0,C 180,E1 8943.493,E2 8943.493} C_VEL
LIN {X 0,Y 602.809,Z 748.488,A -85,B 0,C 180,E1 8945.225,E2 8945.225} C_VEL
LIN {X 0,Y 605.051,Z 705.759,A -85,B 0,C 180,E1 8946.332,E2 8946.332} C_VEL
LIN {X 0,Y 605.63,Z 660.237,A -85,B 0,C 180,E1 8947.055,E2 8947.055} C_VEL
LIN {X 0,Y 579.372,Z 601.31,A -85,B 0,C 180,E1 8949.547,E2 8949.547} C_VEL
LIN {X 0,Y 579.328,Z 601.31,A -85,B 0,C 180,E1 8955.085,E2 8955.085} C_VEL
LIN {X 0,Y 579.284,Z 601.31,A -85,B 0,C 180,E1 8961.123,E2 8961.123} C_VEL
LIN {X 0,Y 579.391,Z 601.31,A -85,B 0,C 180,E1 8966.817,E2 8966.817} C_VEL
LIN {X 0,Y 579.557,Z 601.31,A -85,B 0,C 180,E1 8972.745,E2 8972.745} C_VEL
LIN {X 0,Y 579.69,Z 601.31,A -85,B 0,C 180,E1 8978.538,E2 8978.538} C_VEL
LIN {X 0,Y 579.766,Z 601.31,A -85,B 0,C 180,E1 8983.294,E2 8983.294} C_VEL
LIN {X 0,Y 579.916,Z 601.31,A -85,B 0,C 180,E1 8989.462,E2 8989.462} C_VEL
LIN {X 0,Y 580.109,Z 601.31,A -85,B 0,C 180,E1 8994.002,E2 8994.002} C_VEL
LIN {X 0,Y 580.218,Z 601.31,A -85,B 0,C 180,E1 8998.502,E2 8998.502} C_VEL
LIN {X 0,Y 580.217,Z 601.31,A -85,B 0,C 180,E1 9002.991,E2 9002.991} C_VEL
LIN {X 0,Y 580.055,Z 601.31,A -85,B 0,C 180,E1 9007.501,E2 9007.501} C_VEL
LIN {X 0,Y 579.92,Z 601.31,A -85,B 0,C 180,E1 9012.061,E2 9012.061} C_VEL
LIN {X 0,Y 579.821,Z 601.31,A -85,B 0,C 180,E1 9016.7,E2 9016.7} C_VEL
LIN {X 0,Y 579.699,Z 601.31,A -85,B 0,C 180,E1 9021.458,E2 9021.458} C_VEL
LIN {X 0,Y 579.546,Z 601.31,A -85,B 0,C 180,E1 9027.253,E2 9027.253} C_VEL
LIN {X 0,Y 579.432,Z 601.31,A -85,B 0,C 180,E1 9033.298,E2 9033.298} C_VEL
LIN {X 0,Y 579.325,Z 601.31,A -85,B 0,C 180,E1 9038.869,E2 9038.869} C_VEL
LIN {X 0,Y 579.373,Z 601.31,A -85,B 0,C 180,E1 9045.074,E2 9045.074} C_VEL
LIN {X 0,Y 579.281,Z 601.31,A -85,B 0,C 180,E1 9051.11,E2 9051.11} C_VEL
LIN {X 0,Y 579.409,Z 601.31,A -85,B 0,C 180,E1 9056.784,E2 9056.784} C_VEL
LIN {X 0,Y 579.61,Z 601.651,A -85,B 0,C 180,E1 9060.163,E2 9060.163} C_VEL
LIN {X 0,Y 592.097,Z 638.606,A -85,B 0,C 180,E1 9061.637,E2 9061.637} C_VEL
LIN {X 0,Y 594.877,Z 651.291,A -85,B 0,C 180,E1 9062.15,E2 9062.15} C_VEL
LIN {X 0,Y 592.76,Z 690.658,A -85,B 0,C 180,E1 9063.617,E2 9063.617} C_VEL
LIN {X 0,Y 590.107,Z 727.884,A -85,B 0,C 180,E1 9065.655,E2 9065.655} C_VEL
LIN {X 0,Y 587.498,Z 759.921,A -85,B 0,C 180,E1 9068.036,E2 9068.036} C_VEL
LIN {X 0,Y 585.082,Z 789.106,A -85,B 0,C 180,E1 9070.9,E2 9070.9} C_VEL
LIN {X 0,Y 583.159,Z 814.801,A -85,B 0,C 180,E1 9074.25,E2 9074.25} C_VEL
LIN {X 0,Y 581.941,Z 833.782,A -85,B 0,C 180,E1 9077.606,E2 9077.606} C_VEL
LIN {X 0,Y 581.187,Z 848.511,A -85,B 0,C 180,E1 9081.357,E2 9081.357} C_VEL
LIN {X 0,Y 580.892,Z 856.93,A -85,B 0,C 180,E1 9084.758,E2 9084.758} C_VEL
LIN {X 0,Y 580.658,Z 861.292,A -85,B 0,C 180,E1 9088.501,E2 9088.501} C_VEL
LIN {X 0,Y 580.771,Z 861.222,A -85,B 0,C 180,E1 9091.491,E2 9091.491} C_VEL
LIN {X 0,Y 580.92,Z 856.762,A -85,B 0,C 180,E1 9095.234,E2 9095.234} C_VEL
LIN {X 0,Y 581.2,Z 847.086,A -85,B 0,C 180,E1 9098.995,E2 9098.995} C_VEL
LIN {X 0,Y 582.058,Z 831.454,A -85,B 0,C 180,E1 9102.766,E2 9102.766} C_VEL
LIN {X 0,Y 583.438,Z 810.697,A -85,B 0,C 180,E1 9106.257,E2 9106.257} C_VEL
LIN {X 0,Y 585.472,Z 785.032,A -85,B 0,C 180,E1 9109.46,E2 9109.46} C_VEL
LIN {X 0,Y 588.002,Z 754.646,A -85,B 0,C 180,E1 9112.317,E2 9112.317} C_VEL
LIN {X 0,Y 590.753,Z 719.906,A -85,B 0,C 180,E1 9114.746,E2 9114.746} C_VEL
LIN {X 0,Y 593.169,Z 684.084,A -85,B 0,C 180,E1 9116.576,E2 9116.576} C_VEL
LIN {X 0,Y 594.48,Z 647.459,A -85,B 0,C 180,E1 9117.898,E2 9117.898} C_VEL
LIN {X 0,Y 582.297,Z 609.259,A -85,B 0,C 180,E1 9119.441,E2 9119.441} C_VEL
LIN {X 0,Y 579.501,Z 601.31,A -85,B 0,C 180,E1 9119.783,E2 9119.783} C_VEL
LIN {X 0,Y 579.373,Z 601.31,A -85,B 0,C 180,E1 9125.119,E2 9125.119} C_VEL
LIN {X 0,Y 579.352,Z 601.31,A -85,B 0,C 180,E1 9130.826,E2 9130.826} C_VEL
LIN {X 0,Y 579.379,Z 601.31,A -85,B 0,C 180,E1 9135.096,E2 9135.096} C_VEL
LIN {X 0,Y 579.289,Z 601.31,A -85,B 0,C 180,E1 9141.128,E2 9141.128} C_VEL
LIN {X 0,Y 579.404,Z 601.31,A -85,B 0,C 180,E1 9146.8,E2 9146.8} C_VEL
LIN {X 0,Y 579.595,Z 601.31,A -85,B 0,C 180,E1 9152.719,E2 9152.719} C_VEL
LIN {X 0,Y 579.671,Z 601.31,A -85,B 0,C 180,E1 9157.394,E2 9157.394} C_VEL
LIN {X 0,Y 590.942,Z 640.018,A -85,B 0,C 180,E1 9158.453,E2 9158.453} C_VEL
LIN {X 0,Y 589.665,Z 697.329,A -85,B 0,C 180,E1 9159.411,E2 9159.411} C_VEL
LIN {X 0,Y 588.284,Z 733.921,A -85,B 0,C 180,E1 9160.64,E2 9160.64} C_VEL
LIN {X 0,Y 586.536,Z 766.52,A -85,B 0,C 180,E1 9162.33,E2 9162.33} C_VEL
LIN {X 0,Y 584.775,Z 797.043,A -85,B 0,C 180,E1 9164.604,E2 9164.604} C_VEL
LIN {X 0,Y 583.278,Z 822.72,A -85,B 0,C 180,E1 9167.279,E2 9167.279} C_VEL
LIN {X 0,Y 582.244,Z 843.075,A -85,B 0,C 180,E1 9170.265,E2 9170.265} C_VEL
LIN {X 0,Y 581.719,Z 857.138,A -85,B 0,C 180,E1 9173.272,E2 9173.272} C_VEL
LIN {X 0,Y 581.419,Z 865.879,A -85,B 0,C 180,E1 9176.267,E2 9176.267} C_VEL
LIN {X 0,Y 581.373,Z 869.273,A -85,B 0,C 180,E1 9178.509,E2 9178.509} C_VEL
LIN {X 0,Y 581.415,Z 869.896,A -85,B 0,C 180,E1 9181.495,E2 9181.495} C_VEL
LIN {X 0,Y 581.792,Z 865.914,A -85,B 0,C 180,E1 9184.482,E2 9184.482} C_VEL
LIN {X 0,Y 582.282,Z 857.01,A -85,B 0,C 180,E1 9187.476,E2 9187.476} C_VEL
LIN {X 0,Y 583.209,Z 841.301,A -85,B 0,C 180,E1 9190.667,E2 9190.667} C_VEL
LIN {X 0,Y 584.421,Z 820.614,A -85,B 0,C 180,E1 9193.493,E2 9193.493} C_VEL
LIN {X 0,Y 586.135,Z 794.357,A -85,B 0,C 180,E1 9196.037,E2 9196.037} C_VEL
LIN {X 0,Y 587.823,Z 764.36,A -85,B 0,C 180,E1 9198.113,E2 9198.113} C_VEL
LIN {X 0,Y 589.629,Z 729.601,A -85,B 0,C 180,E1 9199.8,E2 9199.8} C_VEL
LIN {X 0,Y 591.387,Z 690.451,A -85,B 0,C 180,E1 9201.017,E2 9201.017} C_VEL
LIN {X 0,Y 592.594,Z 636.488,A -85,B 0,C 180,E1 9202.058,E2 9202.058} C_VEL
LIN {X 0,Y 579.627,Z 601.31,A -85,B 0,C 180,E1 9203.594,E2 9203.594} C_VEL
LIN {X 0,Y 579.496,Z 601.31,A -85,B 0,C 180,E1 9209.783,E2 9209.783} C_VEL
LIN {X 0,Y 579.386,Z 601.31,A -85,B 0,C 180,E1 9215.117,E2 9215.117} C_VEL
LIN {X 0,Y 579.38,Z 601.31,A -85,B 0,C 180,E1 9220.821,E2 9220.821} C_VEL
LIN {X 0,Y 579.351,Z 601.31,A -85,B 0,C 180,E1 9225.204,E2 9225.204} C_VEL
LIN {X 0,Y 579.217,Z 601.31,A -85,B 0,C 180,E1 9228.576,E2 9228.576} C_VEL
LIN {X 0,Y 575.277,Z 601.31,A -85,B 0,C 180,E1 9229.681,E2 9229.681} C_VEL
LIN {X 0,Y 571.351,Z 601.31,A -85,B 0,C 180,E1 9230.802,E2 9230.802} C_VEL
LIN {X 0,Y 585.141,Z 635.605,A -85,B 0,C 180,E1 9232.229,E2 9232.229} C_VEL
LIN {X 0,Y 595.238,Z 661.659,A -85,B 0,C 180,E1 9233.133,E2 9233.133} C_VEL
LIN {X 0,Y 596.151,Z 670.039,A -85,B 0,C 180,E1 9233.289,E2 9233.289} C_VEL
LIN {X 0,Y 594.956,Z 718.258,A -85,B 0,C 180,E1 9234.094,E2 9234.094} C_VEL
LIN {X 0,Y 592.663,Z 760.274,A -85,B 0,C 180,E1 9235.305,E2 9235.305} C_VEL
LIN {X 0,Y 589.512,Z 804.701,A -85,B 0,C 180,E1 9237.209,E2 9237.209} C_VEL
LIN {X 0,Y 585.911,Z 846.232,A -85,B 0,C 180,E1 9239.661,E2 9239.661} C_VEL
LIN {X 0,Y 582.048,Z 886.311,A -85,B 0,C 180,E1 9242.805,E2 9242.805} C_VEL
LIN {X 0,Y 578.585,Z 921.213,A -85,B 0,C 180,E1 9246.408,E2 9246.408} C_VEL
LIN {X 0,Y 575.91,Z 950.658,A -85,B 0,C 180,E1 9250.399,E2 9250.399} C_VEL
LIN {X 0,Y 574.124,Z 973.049,A -85,B 0,C 180,E1 9254.424,E2 9254.424} C_VEL
LIN {X 0,Y 573.194,Z 988.772,A -85,B 0,C 180,E1 9258.257,E2 9258.257} C_VEL
LIN {X 0,Y 572.647,Z 999.644,A -85,B 0,C 180,E1 9262.402,E2 9262.402} C_VEL
LIN {X 0,Y 572.536,Z 1004.65,A -85,B 0,C 180,E1 9265.45,E2 9265.45} C_VEL
LIN {X 0,Y 572.562,Z 1007.5,A -85,B 0,C 180,E1 9270.004,E2 9270.004} C_VEL
LIN {X 0,Y 572.544,Z 1004.641,A -85,B 0,C 180,E1 9274.558,E2 9274.558} C_VEL
LIN {X 0,Y 572.679,Z 998.06,A -85,B 0,C 180,E1 9278.372,E2 9278.372} C_VEL
LIN {X 0,Y 573.343,Z 985.716,A -85,B 0,C 180,E1 9282.597,E2 9282.597} C_VEL
LIN {X 0,Y 574.508,Z 968.163,A -85,B 0,C 180,E1 9286.616,E2 9286.616} C_VEL
LIN {X 0,Y 576.52,Z 943.432,A -85,B 0,C 180,E1 9290.815,E2 9290.815} C_VEL
LIN {X 0,Y 579.666,Z 913.076,A -85,B 0,C 180,E1 9294.727,E2 9294.727} C_VEL
LIN {X 0,Y 583.526,Z 878.073,A -85,B 0,C 180,E1 9298.211,E2 9298.211} C_VEL
LIN {X 0,Y 587.505,Z 841.159,A -85,B 0,C 180,E1 9301.056,E2 9301.056} C_VEL
LIN {X 0,Y 591.467,Z 802.055,A -85,B 0,C 180,E1 9303.367,E2 9303.367} C_VEL
LIN {X 0,Y 595.094,Z 758.381,A -85,B 0,C 180,E1 9305.259,E2 9305.259} C_VEL
LIN {X 0,Y 598.001,Z 710.988,A -85,B 0,C 180,E1 9306.608,E2 9306.608} C_VEL
LIN {X 0,Y 599.02,Z 663.223,A -85,B 0,C 180,E1 9307.39,E2 9307.39} C_VEL
LIN {X 0,Y 571.492,Z 601.31,A -85,B 0,C 180,E1 9310.064,E2 9310.064} C_VEL
LIN {X 0,Y 571.343,Z 601.31,A -85,B 0,C 180,E1 9315.735,E2 9315.735} C_VEL
LIN {X 0,Y 571.336,Z 601.31,A -85,B 0,C 180,E1 9320.477,E2 9320.477} C_VEL
LIN {X 0,Y 571.399,Z 601.31,A -85,B 0,C 180,E1 9326.167,E2 9326.167} C_VEL
LIN {X 0,Y 571.586,Z 601.31,A -85,B 0,C 180,E1 9331.505,E2 9331.505} C_VEL
LIN {X 0,Y 571.744,Z 601.31,A -85,B 0,C 180,E1 9336.58,E2 9336.58} C_VEL
LIN {X 0,Y 571.819,Z 601.31,A -85,B 0,C 180,E1 9342.554,E2 9342.554} C_VEL
LIN {X 0,Y 571.947,Z 601.31,A -85,B 0,C 180,E1 9348.602,E2 9348.602} C_VEL
LIN {X 0,Y 572.211,Z 601.31,A -85,B 0,C 180,E1 9353.919,E2 9353.919} C_VEL
LIN {X 0,Y 572.316,Z 601.31,A -85,B 0,C 180,E1 9358.481,E2 9358.481} C_VEL
LIN {X 0,Y 572.317,Z 601.31,A -85,B 0,C 180,E1 9363.033,E2 9363.033} C_VEL
LIN {X 0,Y 572.137,Z 601.31,A -85,B 0,C 180,E1 9367.606,E2 9367.606} C_VEL
LIN {X 0,Y 571.998,Z 601.31,A -85,B 0,C 180,E1 9372.23,E2 9372.23} C_VEL
LIN {X 0,Y 571.849,Z 601.31,A -85,B 0,C 180,E1 9377.455,E2 9377.455} C_VEL
LIN {X 0,Y 571.735,Z 601.31,A -85,B 0,C 180,E1 9383.416,E2 9383.416} C_VEL
LIN {X 0,Y 571.562,Z 601.31,A -85,B 0,C 180,E1 9388.967,E2 9388.967} C_VEL
LIN {X 0,Y 571.43,Z 601.31,A -85,B 0,C 180,E1 9394.707,E2 9394.707} C_VEL
LIN {X 0,Y 571.366,Z 601.31,A -85,B 0,C 180,E1 9399.725,E2 9399.725} C_VEL
LIN {X 0,Y 571.378,Z 601.31,A -85,B 0,C 180,E1 9405.71,E2 9405.71} C_VEL
LIN {X 0,Y 571.327,Z 601.31,A -85,B 0,C 180,E1 9410.463,E2 9410.463} C_VEL
LIN {X 0,Y 571.421,Z 601.31,A -85,B 0,C 180,E1 9416.157,E2 9416.157} C_VEL
LIN {X 0,Y 571.67,Z 601.31,A -85,B 0,C 180,E1 9419.688,E2 9419.688} C_VEL
LIN {X 0,Y 584.669,Z 639.206,A -85,B 0,C 180,E1 9421.266,E2 9421.266} C_VEL
LIN {X 0,Y 587.791,Z 652.768,A -85,B 0,C 180,E1 9421.835,E2 9421.835} C_VEL
LIN {X 0,Y 585.632,Z 691.425,A -85,B 0,C 180,E1 9423.298,E2 9423.298} C_VEL
LIN {X 0,Y 582.921,Z 728.096,A -85,B 0,C 180,E1 9425.318,E2 9425.318} C_VEL
LIN {X 0,Y 580.102,Z 760.926,A -85,B 0,C 180,E1 9427.784,E2 9427.784} C_VEL
LIN {X 0,Y 577.551,Z 790.047,A -85,B 0,C 180,E1 9430.686,E2 9430.686} C_VEL
LIN {X 0,Y 575.486,Z 815.623,A -85,B 0,C 180,E1 9434.074,E2 9434.074} C_VEL
LIN {X 0,Y 574.049,Z 836.062,A -85,B 0,C 180,E1 9437.805,E2 9437.805} C_VEL
LIN {X 0,Y 573.344,Z 850.48,A -85,B 0,C 180,E1 9441.638,E2 9441.638} C_VEL
LIN {X 0,Y 572.996,Z 859.086,A -85,B 0,C 180,E1 9445.446,E2 9445.446} C_VEL
LIN {X 0,Y 572.828,Z 862.272,A -85,B 0,C 180,E1 9448.48,E2 9448.48} C_VEL
LIN {X 0,Y 572.949,Z 862.201,A -85,B 0,C 180,E1 9451.511,E2 9451.511} C_VEL
LIN {X 0,Y 573.095,Z 857.667,A -85,B 0,C 180,E1 9455.305,E2 9455.305} C_VEL
LIN {X 0,Y 573.388,Z 847.844,A -85,B 0,C 180,E1 9459.119,E2 9459.119} C_VEL
LIN {X 0,Y 574.257,Z 833.221,A -85,B 0,C 180,E1 9462.705,E2 9462.705} C_VEL
LIN {X 0,Y 575.7,Z 812.421,A -85,B 0,C 180,E1 9466.311,E2 9466.311} C_VEL
LIN {X 0,Y 577.774,Z 787.816,A -85,B 0,C 180,E1 9469.474,E2 9469.474} C_VEL
LIN {X 0,Y 580.467,Z 757.091,A -85,B 0,C 180,E1 9472.458,E2 9472.458} C_VEL
LIN {X 0,Y 583.418,Z 722.195,A -85,B 0,C 180,E1 9474.958,E2 9474.958} C_VEL
LIN {X 0,Y 585.938,Z 686.772,A -85,B 0,C 180,E1 9476.815,E2 9476.815} C_VEL
LIN {X 0,Y 587.222,Z 648.998,A -85,B 0,C 180,E1 9478.224,E2 9478.224} C_VEL
LIN {X 0,Y 575.99,Z 613.21,A -85,B 0,C 180,E1 9479.71,E2 9479.71} C_VEL
LIN {X 0,Y 571.59,Z 601.31,A -85,B 0,C 180,E1 9480.238,E2 9480.238} C_VEL
LIN {X 0,Y 571.473,Z 601.31,A -85,B 0,C 180,E1 9485.678,E2 9485.678} C_VEL
LIN {X 0,Y 571.376,Z 601.31,A -85,B 0,C 180,E1 9491.521,E2 9491.521} C_VEL
LIN {X 0,Y 571.371,Z 601.31,A -85,B 0,C 180,E1 9496.425,E2 9496.425} C_VEL
LIN {X 0,Y 571.41,Z 601.31,A -85,B 0,C 180,E1 9502.696,E2 9502.696} C_VEL
LIN {X 0,Y 571.524,Z 601.31,A -85,B 0,C 180,E1 9508.027,E2 9508.027} C_VEL
LIN {X 0,Y 571.686,Z 601.31,A -85,B 0,C 180,E1 9513.228,E2 9513.228} C_VEL
LIN {X 0,Y 571.758,Z 601.31,A -85,B 0,C 180,E1 9517.072,E2 9517.072} C_VEL
LIN {X 0,Y 583.604,Z 641.581,A -85,B 0,C 180,E1 9518.191,E2 9518.191} C_VEL
LIN {X 0,Y 582.287,Z 696.718,A -85,B 0,C 180,E1 9519.13,E2 9519.13} C_VEL
LIN {X 0,Y 580.859,Z 732.73,A -85,B 0,C 180,E1 9520.332,E2 9520.332} C_VEL
LIN {X 0,Y 578.993,Z 766.713,A -85,B 0,C 180,E1 9522.098,E2 9522.098} C_VEL
LIN {X 0,Y 577.142,Z 797.333,A -85,B 0,C 180,E1 9524.395,E2 9524.395} C_VEL
LIN {X 0,Y 575.607,Z 822.704,A -85,B 0,C 180,E1 9527.047,E2 9527.047} C_VEL
LIN {X 0,Y 574.531,Z 842.672,A -85,B 0,C 180,E1 9529.942,E2 9529.942} C_VEL
LIN {X 0,Y 573.911,Z 857.931,A -85,B 0,C 180,E1 9533.18,E2 9533.18} C_VEL
LIN {X 0,Y 573.605,Z 866.803,A -85,B 0,C 180,E1 9536.216,E2 9536.216} C_VEL
LIN {X 0,Y 573.559,Z 870.278,A -85,B 0,C 180,E1 9538.488,E2 9538.488} C_VEL
LIN {X 0,Y 573.597,Z 870.984,A -85,B 0,C 180,E1 9541.515,E2 9541.515} C_VEL
LIN {X 0,Y 574.017,Z 867.041,A -85,B 0,C 180,E1 9544.543,E2 9544.543} C_VEL
LIN {X 0,Y 574.577,Z 857.138,A -85,B 0,C 180,E1 9547.837,E2 9547.837} C_VEL
LIN {X 0,Y 575.642,Z 841.344,A -85,B 0,C 180,E1 9551.001,E2 9551.001} C_VEL
LIN {X 0,Y 576.963,Z 820.144,A -85,B 0,C 180,E1 9553.864,E2 9553.864} C_VEL
LIN {X 0,Y 578.799,Z 793.16,A -85,B 0,C 180,E1 9556.441,E2 9556.441} C_VEL
LIN {X 0,Y 580.666,Z 762.527,A -85,B 0,C 180,E1 9558.541,E2 9558.541} C_VEL
LIN {X 0,Y 582.666,Z 725.711,A -85,B 0,C 180,E1 9560.282,E2 9560.282} C_VEL
LIN {X 0,Y 584.505,Z 686.521,A -85,B 0,C 180,E1 9561.452,E2 9561.452} C_VEL
LIN {X 0,Y 585.764,Z 638.706,A -85,B 0,C 180,E1 9562.388,E2 9562.388} C_VEL
LIN {X 0,Y 572.841,Z 605.439,A -85,B 0,C 180,E1 9563.94,E2 9563.94} C_VEL
LIN {X 0,Y 571.66,Z 601.31,A -85,B 0,C 180,E1 9564.156,E2 9564.156} C_VEL
LIN {X 0,Y 571.602,Z 601.31,A -85,B 0,C 180,E1 9570.237,E2 9570.237} C_VEL
LIN {X 0,Y 571.49,Z 601.31,A -85,B 0,C 180,E1 9575.676,E2 9575.676} C_VEL
LIN {X 0,Y 571.396,Z 601.31,A -85,B 0,C 180,E1 9581.516,E2 9581.516} C_VEL
LIN {X 0,Y 571.367,Z 601.31,A -85,B 0,C 180,E1 9586.416,E2 9586.416} C_VEL
LIN {X 0,Y 571.351,Z 601.31,A -85,B 0,C 180,E1 9590.802,E2 9590.802} C_VEL
LIN {X 0,Y 574.944,Z 606.384,A -85,B 0,C 180,E1 9591.168,E2 9591.168} C_VEL
LIN {X 0,Y 576.352,Z 619.439,A -85,B 0,C 180,E1 9591.409,E2 9591.409} C_VEL
LIN {X 0,Y 576.96,Z 633.536,A -85,B 0,C 180,E1 9591.704,E2 9591.704} C_VEL
LIN {X 0,Y 577.355,Z 634.702,A -85,B 0,C 180,E1 9591.747,E2 9591.747} C_VEL
LIN {X 0,Y 588.763,Z 665.034,A -85,B 0,C 180,E1 9592.831,E2 9592.831} C_VEL
LIN {X 0,Y 588.099,Z 714.836,A -85,B 0,C 180,E1 9593.665,E2 9593.665} C_VEL
LIN {X 0,Y 585.524,Z 759.602,A -85,B 0,C 180,E1 9594.948,E2 9594.948} C_VEL
LIN {X 0,Y 582.232,Z 804.092,A -85,B 0,C 180,E1 9596.877,E2 9596.877} C_VEL
LIN {X 0,Y 578.327,Z 846.957,A -85,B 0,C 180,E1 9599.455,E2 9599.455} C_VEL
LIN {X 0,Y 574.428,Z 885.917,A -85,B 0,C 180,E1 9602.567,E2 9602.567} C_VEL
LIN {X 0,Y 570.963,Z 919.567,A -85,B 0,C 180,E1 9606.074,E2 9606.074} C_VEL
LIN {X 0,Y 568.201,Z 948.011,A -85,B 0,C 180,E1 9609.924,E2 9609.924} C_VEL
LIN {X 0,Y 566.417,Z 970.489,A -85,B 0,C 180,E1 9613.912,E2 9613.912} C_VEL
LIN {X 0,Y 565.323,Z 988.281,A -85,B 0,C 180,E1 9618.212,E2 9618.212} C_VEL
LIN {X 0,Y 564.781,Z 999.552,A -85,B 0,C 180,E1 9622.295,E2 9622.295} C_VEL
LIN {X 0,Y 564.642,Z 1004.65,A -85,B 0,C 180,E1 9625.387,E2 9625.387} C_VEL
LIN {X 0,Y 564.662,Z 1007.5,A -85,B 0,C 180,E1 9630.004,E2 9630.004} C_VEL
LIN {X 0,Y 564.651,Z 1004.641,A -85,B 0,C 180,E1 9634.622,E2 9634.622} C_VEL
LIN {X 0,Y 564.805,Z 997.865,A -85,B 0,C 180,E1 9638.489,E2 9638.489} C_VEL
LIN {X 0,Y 565.48,Z 984.821,A -85,B 0,C 180,E1 9642.776,E2 9642.776} C_VEL
LIN {X 0,Y 566.626,Z 966.983,A -85,B 0,C 180,E1 9646.891,E2 9646.891} C_VEL
LIN {X 0,Y 568.779,Z 942.997,A -85,B 0,C 180,E1 9651.015,E2 9651.015} C_VEL
LIN {X 0,Y 572.166,Z 911.916,A -85,B 0,C 180,E1 9655.074,E2 9655.074} C_VEL
LIN {X 0,Y 576.331,Z 875.905,A -85,B 0,C 180,E1 9658.677,E2 9658.677} C_VEL
LIN {X 0,Y 580.736,Z 836.869,A -85,B 0,C 180,E1 9661.662,E2 9661.662} C_VEL
LIN {X 0,Y 584.828,Z 796.958,A -85,B 0,C 180,E1 9663.966,E2 9663.966} C_VEL
LIN {X 0,Y 588.318,Z 755.77,A -85,B 0,C 180,E1 9665.716,E2 9665.716} C_VEL
LIN {X 0,Y 591.15,Z 710.904,A -85,B 0,C 180,E1 9666.99,E2 9666.99} C_VEL
LIN {X 0,Y 592.222,Z 665.792,A -85,B 0,C 180,E1 9667.742,E2 9667.742} C_VEL
LIN {X 0,Y 563.558,Z 601.31,A -85,B 0,C 180,E1 9670.535,E2 9670.535} C_VEL
LIN {X 0,Y 563.44,Z 601.31,A -85,B 0,C 180,E1 9676.565,E2 9676.565} C_VEL
LIN {X 0,Y 563.385,Z 601.31,A -85,B 0,C 180,E1 9681.795,E2 9681.795} C_VEL
LIN {X 0,Y 563.523,Z 601.31,A -85,B 0,C 180,E1 9687.474,E2 9687.474} C_VEL
LIN {X 0,Y 563.694,Z 601.31,A -85,B 0,C 180,E1 9692.813,E2 9692.813} C_VEL
LIN {X 0,Y 563.844,Z 601.31,A -85,B 0,C 180,E1 9697.903,E2 9697.903} C_VEL
LIN {X 0,Y 563.943,Z 601.31,A -85,B 0,C 180,E1 9702.811,E2 9702.811} C_VEL
LIN {X 0,Y 564.033,Z 601.31,A -85,B 0,C 180,E1 9707.59,E2 9707.59} C_VEL
LIN {X 0,Y 564.292,Z 601.31,A -85,B 0,C 180,E1 9713.502,E2 9713.502} C_VEL
LIN {X 0,Y 564.415,Z 601.31,A -85,B 0,C 180,E1 9718.46,E2 9718.46} C_VEL
LIN {X 0,Y 564.413,Z 601.31,A -85,B 0,C 180,E1 9723.075,E2 9723.075} C_VEL
LIN {X 0,Y 564.242,Z 601.31,A -85,B 0,C 180,E1 9727.713,E2 9727.713} C_VEL
LIN {X 0,Y 564.073,Z 601.31,A -85,B 0,C 180,E1 9732.405,E2 9732.405} C_VEL
LIN {X 0,Y 563.984,Z 601.31,A -85,B 0,C 180,E1 9737.183,E2 9737.183} C_VEL
LIN {X 0,Y 563.846,Z 601.31,A -85,B 0,C 180,E1 9742.093,E2 9742.093} C_VEL
LIN {X 0,Y 563.654,Z 601.31,A -85,B 0,C 180,E1 9747.48,E2 9747.48} C_VEL
LIN {X 0,Y 563.537,Z 601.31,A -85,B 0,C 180,E1 9752.52,E2 9752.52} C_VEL
LIN {X 0,Y 563.435,Z 601.31,A -85,B 0,C 180,E1 9758.196,E2 9758.196} C_VEL
LIN {X 0,Y 563.498,Z 601.31,A -85,B 0,C 180,E1 9764.342,E2 9764.342} C_VEL
LIN {X 0,Y 563.388,Z 601.31,A -85,B 0,C 180,E1 9769.794,E2 9769.794} C_VEL
LIN {X 0,Y 563.491,Z 601.31,A -85,B 0,C 180,E1 9775.615,E2 9775.615} C_VEL
LIN {X 0,Y 563.716,Z 601.31,A -85,B 0,C 180,E1 9779.223,E2 9779.223} C_VEL
LIN {X 0,Y 577.096,Z 639.184,A -85,B 0,C 180,E1 9780.855,E2 9780.855} C_VEL
LIN {X 0,Y 580.712,Z 654.377,A -85,B 0,C 180,E1 9781.512,E2 9781.512} C_VEL
LIN {X 0,Y 578.432,Z 693.576,A -85,B 0,C 180,E1 9783.027,E2 9783.027} C_VEL
LIN {X 0,Y 575.494,Z 731.193,A -85,B 0,C 180,E1 9785.16,E2 9785.16} C_VEL
LIN {X 0,Y 572.534,Z 764.067,A -85,B 0,C 180,E1 9787.709,E2 9787.709} C_VEL
LIN {X 0,Y 569.826,Z 793.294,A -85,B 0,C 180,E1 9790.72,E2 9790.72} C_VEL
LIN {X 0,Y 567.624,Z 818.79,A -85,B 0,C 180,E1 9794.251,E2 9794.251} C_VEL
LIN {X 0,Y 566.206,Z 838.543,A -85,B 0,C 180,E1 9798.026,E2 9798.026} C_VEL
LIN {X 0,Y 565.472,Z 852.44,A -85,B 0,C 180,E1 9801.909,E2 9801.909} C_VEL
LIN {X 0,Y 565.179,Z 860.011,A -85,B 0,C 180,E1 9805.383,E2 9805.383} C_VEL
LIN {X 0,Y 565.007,Z 863.248,A -85,B 0,C 180,E1 9808.459,E2 9808.459} C_VEL
LIN {X 0,Y 565.126,Z 863.18,A -85,B 0,C 180,E1 9811.532,E2 9811.532} C_VEL
LIN {X 0,Y 565.268,Z 858.574,A -85,B 0,C 180,E1 9815.379,E2 9815.379} C_VEL
LIN {X 0,Y 565.6,Z 848.649,A -85,B 0,C 180,E1 9819.245,E2 9819.245} C_VEL
LIN {X 0,Y 566.504,Z 834.712,A -85,B 0,C 180,E1 9822.73,E2 9822.73} C_VEL
LIN {X 0,Y 568.011,Z 814.24,A -85,B 0,C 180,E1 9826.369,E2 9826.369} C_VEL
LIN {X 0,Y 570.225,Z 789.158,A -85,B 0,C 180,E1 9829.664,E2 9829.664} C_VEL
LIN {X 0,Y 573.032,Z 758.94,A -85,B 0,C 180,E1 9832.654,E2 9832.654} C_VEL
LIN {X 0,Y 576.154,Z 724.288,A -85,B 0,C 180,E1 9835.191,E2 9835.191} C_VEL
LIN {X 0,Y 578.774,Z 688.974,A -85,B 0,C 180,E1 9837.085,E2 9837.085} C_VEL
LIN {X 0,Y 580.166,Z 651.168,A -85,B 0,C 180,E1 9838.531,E2 9838.531} C_VEL
LIN {X 0,Y 569.554,Z 616.841,A -85,B 0,C 180,E1 9839.999,E2 9839.999} C_VEL
LIN {X 0,Y 563.639,Z 601.31,A -85,B 0,C 180,E1 9840.71,E2 9840.71} C_VEL
LIN {X 0,Y 563.532,Z 601.31,A -85,B 0,C 180,E1 9846.26,E2 9846.26} C_VEL
LIN {X 0,Y 563.487,Z 601.31,A -85,B 0,C 180,E1 9852.235,E2 9852.235} C_VEL
LIN {X 0,Y 563.434,Z 601.31,A -85,B 0,C 180,E1 9857.768,E2 9857.768} C_VEL
LIN {X 0,Y 563.468,Z 601.31,A -85,B 0,C 180,E1 9863.769,E2 9863.769} C_VEL
LIN {X 0,Y 563.644,Z 601.31,A -85,B 0,C 180,E1 9869.334,E2 9869.334} C_VEL
LIN {X 0,Y 563.755,Z 601.31,A -85,B 0,C 180,E1 9874.538,E2 9874.538} C_VEL
LIN {X 0,Y 563.839,Z 601.31,A -85,B 0,C 180,E1 9876.719,E2 9876.719} C_VEL
LIN {X 0,Y 576.209,Z 641.965,A -85,B 0,C 180,E1 9877.917,E2 9877.917} C_VEL
LIN {X 0,Y 574.858,Z 697.087,A -85,B 0,C 180,E1 9878.876,E2 9878.876} C_VEL
LIN {X 0,Y 573.339,Z 733.511,A -85,B 0,C 180,E1 9880.114,E2 9880.114} C_VEL
LIN {X 0,Y 571.419,Z 766.653,A -85,B 0,C 180,E1 9881.853,E2 9881.853} C_VEL
LIN {X 0,Y 569.545,Z 796.408,A -85,B 0,C 180,E1 9884.082,E2 9884.082} C_VEL
LIN {X 0,Y 568.039,Z 821.315,A -85,B 0,C 180,E1 9886.645,E2 9886.645} C_VEL
LIN {X 0,Y 566.839,Z 842.145,A -85,B 0,C 180,E1 9889.609,E2 9889.609} C_VEL
LIN {X 0,Y 566.142,Z 857.235,A -85,B 0,C 180,E1 9892.7,E2 9892.7} C_VEL
LIN {X 0,Y 565.779,Z 867.721,A -85,B 0,C 180,E1 9896.164,E2 9896.164} C_VEL
LIN {X 0,Y 565.738,Z 871.279,A -85,B 0,C 180,E1 9898.468,E2 9898.468} C_VEL
LIN {X 0,Y 565.776,Z 872.064,A -85,B 0,C 180,E1 9901.536,E2 9901.536} C_VEL
LIN {X 0,Y 566.233,Z 868.182,A -85,B 0,C 180,E1 9904.606,E2 9904.606} C_VEL
LIN {X 0,Y 566.876,Z 858.085,A -85,B 0,C 180,E1 9908.006,E2 9908.006} C_VEL
LIN {X 0,Y 567.98,Z 842.547,A -85,B 0,C 180,E1 9911.151,E2 9911.151} C_VEL
LIN {X 0,Y 569.39,Z 821.365,A -85,B 0,C 180,E1 9914.052,E2 9914.052} C_VEL
LIN {X 0,Y 571.346,Z 794.464,A -85,B 0,C 180,E1 9916.662,E2 9916.662} C_VEL
LIN {X 0,Y 573.307,Z 763.947,A -85,B 0,C 180,E1 9918.788,E2 9918.788} C_VEL
LIN {X 0,Y 575.427,Z 727.61,A -85,B 0,C 180,E1 9920.548,E2 9920.548} C_VEL
LIN {X 0,Y 577.508,Z 686.797,A -85,B 0,C 180,E1 9921.807,E2 9921.807} C_VEL
LIN {X 0,Y 578.812,Z 640.603,A -85,B 0,C 180,E1 9922.745,E2 9922.745} C_VEL
LIN {X 0,Y 565.699,Z 606.589,A -85,B 0,C 180,E1 9924.411,E2 9924.411} C_VEL
LIN {X 0,Y 563.731,Z 601.31,A -85,B 0,C 180,E1 9924.708,E2 9924.708} C_VEL
LIN {X 0,Y 563.666,Z 601.31,A -85,B 0,C 180,E1 9930.708,E2 9930.708} C_VEL
LIN {X 0,Y 563.56,Z 601.31,A -85,B 0,C 180,E1 9936.257,E2 9936.257} C_VEL
LIN {X 0,Y 563.501,Z 601.31,A -85,B 0,C 180,E1 9942.231,E2 9942.231} C_VEL
LIN {X 0,Y 563.432,Z 601.31,A -85,B 0,C 180,E1 9947.76,E2 9947.76} C_VEL
LIN {X 0,Y 563.46,Z 602.006,A -85,B 0,C 180,E1 9950.294,E2 9950.294} C_VEL
LIN {X 0,Y 577.355,Z 634.702,A -85,B 0,C 180,E1 9951.747,E2 9951.747} C_VEL
LIN {X 0,Y 579.179,Z 642.897,A -85,B 0,C 180,E1 9951.975,E2 9951.975} C_VEL
LIN {X 0,Y 580.93,Z 664.371,A -85,B 0,C 180,E1 9952.379,E2 9952.379} C_VEL
LIN {X 0,Y 582.25,Z 668.285,A -85,B 0,C 180,E1 9952.509,E2 9952.509} C_VEL
LIN {X 0,Y 581.023,Z 717.375,A -85,B 0,C 180,E1 9953.357,E2 9953.357} C_VEL
LIN {X 0,Y 578.348,Z 760.413,A -85,B 0,C 180,E1 9954.633,E2 9954.633} C_VEL
LIN {X 0,Y 575.026,Z 803.128,A -85,B 0,C 180,E1 9956.513,E2 9956.513} C_VEL
LIN {X 0,Y 571.006,Z 845.288,A -85,B 0,C 180,E1 9959.066,E2 9959.066} C_VEL
LIN {X 0,Y 566.953,Z 884.399,A -85,B 0,C 180,E1 9962.215,E2 9962.215} C_VEL
LIN {X 0,Y 563.135,Z 920.129,A -85,B 0,C 180,E1 9965.991,E2 9965.991} C_VEL
LIN {X 0,Y 560.283,Z 949.239,A -85,B 0,C 180,E1 9970.041,E2 9970.041} C_VEL
LIN {X 0,Y 558.411,Z 972.029,A -85,B 0,C 180,E1 9974.26,E2 9974.26} C_VEL
LIN {X 0,Y 557.386,Z 988.82,A -85,B 0,C 180,E1 9978.539,E2 9978.539} C_VEL
LIN {X 0,Y 556.871,Z 1000.139,A -85,B 0,C 180,E1 9982.894,E2 9982.894} C_VEL
LIN {X 0,Y 556.712,Z 1005.719,A -85,B 0,C 180,E1 9986.884,E2 9986.884} C_VEL
LIN {X 0,Y 556.771,Z 1007.107,A -85,B 0,C 180,E1 9990.004,E2 9990.004} C_VEL
LIN {X 0,Y 556.8,Z 1004.055,A -85,B 0,C 180,E1 9994.687,E2 9994.687} C_VEL
LIN {X 0,Y 556.992,Z 995.993,A -85,B 0,C 180,E1 9999.003,E2 9999.003} C_VEL
LIN {X 0,Y 557.708,Z 982.49,A -85,B 0,C 180,E1 10003.356,E2 10003.356} C_VEL
LIN {X 0,Y 558.881,Z 964.866,A -85,B 0,C 180,E1 10007.356,E2 10007.356} C_VEL
LIN {X 0,Y 561.179,Z 940.954,A -85,B 0,C 180,E1 10011.464,E2 10011.464} C_VEL
LIN {X 0,Y 564.635,Z 910.749,A -85,B 0,C 180,E1 10015.432,E2 10015.432} C_VEL
LIN {X 0,Y 569.002,Z 874.548,A -85,B 0,C 180,E1 10019.082,E2 10019.082} C_VEL
LIN {X 0,Y 573.796,Z 833.91,A -85,B 0,C 180,E1 10022.187,E2 10022.187} C_VEL
LIN {X 0,Y 578.363,Z 790.955,A -85,B 0,C 180,E1 10024.617,E2 10024.617} C_VEL
LIN {X 0,Y 582.108,Z 747.273,A -85,B 0,C 180,E1 10026.37,E2 10026.37} C_VEL
LIN {X 0,Y 584.7,Z 703.22,A -85,B 0,C 180,E1 10027.526,E2 10027.526} C_VEL
LIN {X 0,Y 585.322,Z 668.078,A -85,B 0,C 180,E1 10028.111,E2 10028.111} C_VEL
LIN {X 0,Y 555.612,Z 601.31,A -85,B 0,C 180,E1 10031.073,E2 10031.073} C_VEL
LIN {X 0,Y 555.518,Z 601.31,A -85,B 0,C 180,E1 10037.435,E2 10037.435} C_VEL
LIN {X 0,Y 555.455,Z 601.31,A -85,B 0,C 180,E1 10043.128,E2 10043.128} C_VEL
LIN {X 0,Y 555.641,Z 601.31,A -85,B 0,C 180,E1 10048.799,E2 10048.799} C_VEL
LIN {X 0,Y 555.814,Z 601.31,A -85,B 0,C 180,E1 10054.144,E2 10054.144} C_VEL
LIN {X 0,Y 555.925,Z 601.31,A -85,B 0,C 180,E1 10059.251,E2 10059.251} C_VEL
LIN {X 0,Y 556.033,Z 601.31,A -85,B 0,C 180,E1 10064.188,E2 10064.188} C_VEL
LIN {X 0,Y 556.177,Z 601.31,A -85,B 0,C 180,E1 10069.007,E2 10069.007} C_VEL
LIN {X 0,Y 556.412,Z 601.31,A -85,B 0,C 180,E1 10073.746,E2 10073.746} C_VEL
LIN {X 0,Y 556.52,Z 601.31,A -85,B 0,C 180,E1 10078.438,E2 10078.438} C_VEL
LIN {X 0,Y 556.517,Z 601.31,A -85,B 0,C 180,E1 10083.119,E2 10083.119} C_VEL
LIN {X 0,Y 556.322,Z 601.31,A -85,B 0,C 180,E1 10087.823,E2 10087.823} C_VEL
LIN {X 0,Y 556.177,Z 601.31,A -85,B 0,C 180,E1 10092.584,E2 10092.584} C_VEL
LIN {X 0,Y 556.041,Z 601.31,A -85,B 0,C 180,E1 10097.48,E2 10097.48} C_VEL
LIN {X 0,Y 555.914,Z 601.31,A -85,B 0,C 180,E1 10102.425,E2 10102.425} C_VEL
LIN {X 0,Y 555.772,Z 601.31,A -85,B 0,C 180,E1 10107.603,E2 10107.603} C_VEL
LIN {X 0,Y 555.627,Z 601.31,A -85,B 0,C 180,E1 10113.042,E2 10113.042} C_VEL
LIN {X 0,Y 555.538,Z 601.31,A -85,B 0,C 180,E1 10118.84,E2 10118.84} C_VEL
LIN {X 0,Y 555.58,Z 601.31,A -85,B 0,C 180,E1 10124.833,E2 10124.833} C_VEL
LIN {X 0,Y 555.517,Z 601.31,A -85,B 0,C 180,E1 10129.775,E2 10129.775} C_VEL
LIN {X 0,Y 555.519,Z 601.31,A -85,B 0,C 180,E1 10135.05,E2 10135.05} C_VEL
LIN {X 0,Y 555.753,Z 601.362,A -85,B 0,C 180,E1 10138.736,E2 10138.736} C_VEL
LIN {X 0,Y 570.008,Z 640.668,A -85,B 0,C 180,E1 10140.499,E2 10140.499} C_VEL
LIN {X 0,Y 573.662,Z 656.991,A -85,B 0,C 180,E1 10141.214,E2 10141.214} C_VEL
LIN {X 0,Y 571.22,Z 696.484,A -85,B 0,C 180,E1 10142.786,E2 10142.786} C_VEL
LIN {X 0,Y 568.236,Z 732.859,A -85,B 0,C 180,E1 10144.899,E2 10144.899} C_VEL
LIN {X 0,Y 565.159,Z 765.318,A -85,B 0,C 180,E1 10147.457,E2 10147.457} C_VEL
LIN {X 0,Y 562.285,Z 794.812,A -85,B 0,C 180,E1 10150.548,E2 10150.548} C_VEL
LIN {X 0,Y 559.978,Z 820.072,A -85,B 0,C 180,E1 10154.113,E2 10154.113} C_VEL
LIN {X 0,Y 558.521,Z 838.73,A -85,B 0,C 180,E1 10157.707,E2 10157.707} C_VEL
LIN {X 0,Y 557.749,Z 852.204,A -85,B 0,C 180,E1 10161.403,E2 10161.403} C_VEL
LIN {X 0,Y 557.35,Z 860.966,A -85,B 0,C 180,E1 10165.318,E2 10165.318} C_VEL
LIN {X 0,Y 557.17,Z 864.23,A -85,B 0,C 180,E1 10168.437,E2 10168.437} C_VEL
LIN {X 0,Y 557.307,Z 864.16,A -85,B 0,C 180,E1 10171.554,E2 10171.554} C_VEL
LIN {X 0,Y 557.44,Z 859.514,A -85,B 0,C 180,E1 10175.455,E2 10175.455} C_VEL
LIN {X 0,Y 557.828,Z 849.528,A -85,B 0,C 180,E1 10179.375,E2 10179.375} C_VEL
LIN {X 0,Y 558.798,Z 835.471,A -85,B 0,C 180,E1 10182.922,E2 10182.922} C_VEL
LIN {X 0,Y 560.454,Z 814.684,A -85,B 0,C 180,E1 10186.648,E2 10186.648} C_VEL
LIN {X 0,Y 562.862,Z 789.194,A -85,B 0,C 180,E1 10190.017,E2 10190.017} C_VEL
LIN {X 0,Y 565.891,Z 758.406,A -85,B 0,C 180,E1 10193.062,E2 10193.062} C_VEL
LIN {X 0,Y 568.987,Z 724.856,A -85,B 0,C 180,E1 10195.531,E2 10195.531} C_VEL
LIN {X 0,Y 571.754,Z 688.954,A -85,B 0,C 180,E1 10197.467,E2 10197.467} C_VEL
LIN {X 0,Y 573.257,Z 653.574,A -85,B 0,C 180,E1 10198.832,E2 10198.832} C_VEL
LIN {X 0,Y 563.086,Z 620.304,A -85,B 0,C 180,E1 10200.301,E2 10200.301} C_VEL
LIN {X 0,Y 555.661,Z 601.31,A -85,B 0,C 180,E1 10201.2,E2 10201.2} C_VEL
LIN {X 0,Y 555.541,Z 601.31,A -85,B 0,C 180,E1 10206.867,E2 10206.867} C_VEL
LIN {X 0,Y 555.577,Z 601.31,A -85,B 0,C 180,E1 10212.98,E2 10212.98} C_VEL
LIN {X 0,Y 555.504,Z 601.31,A -85,B 0,C 180,E1 10219.122,E2 10219.122} C_VEL
LIN {X 0,Y 555.519,Z 601.31,A -85,B 0,C 180,E1 10225.066,E2 10225.066} C_VEL
LIN {X 0,Y 555.734,Z 601.31,A -85,B 0,C 180,E1 10230.739,E2 10230.739} C_VEL
LIN {X 0,Y 555.943,Z 602.112,A -85,B 0,C 180,E1 10236.416,E2 10236.416} C_VEL
LIN {X 0,Y 568.815,Z 643.692,A -85,B 0,C 180,E1 10237.66,E2 10237.66} C_VEL
LIN {X 0,Y 567.418,Z 697.667,A -85,B 0,C 180,E1 10238.62,E2 10238.62} C_VEL
LIN {X 0,Y 565.798,Z 734.287,A -85,B 0,C 180,E1 10239.889,E2 10239.889} C_VEL
LIN {X 0,Y 563.77,Z 768.107,A -85,B 0,C 180,E1 10241.699,E2 10241.699} C_VEL
LIN {X 0,Y 561.815,Z 798.154,A -85,B 0,C 180,E1 10243.999,E2 10243.999} C_VEL
LIN {X 0,Y 560.17,Z 823.744,A -85,B 0,C 180,E1 10246.709,E2 10246.709} C_VEL
LIN {X 0,Y 558.923,Z 844.97,A -85,B 0,C 180,E1 10249.855,E2 10249.855} C_VEL
LIN {X 0,Y 558.294,Z 859.492,A -85,B 0,C 180,E1 10252.988,E2 10252.988} C_VEL
LIN {X 0,Y 557.953,Z 868.636,A -85,B 0,C 180,E1 10256.11,E2 10256.11} C_VEL
LIN {X 0,Y 557.915,Z 872.267,A -85,B 0,C 180,E1 10258.446,E2 10258.446} C_VEL
LIN {X 0,Y 557.971,Z 873.151,A -85,B 0,C 180,E1 10261.558,E2 10261.558} C_VEL
LIN {X 0,Y 558.437,Z 869.345,A -85,B 0,C 180,E1 10264.67,E2 10264.67} C_VEL
LIN {X 0,Y 559.057,Z 860.574,A -85,B 0,C 180,E1 10267.789,E2 10267.789} C_VEL
LIN {X 0,Y 560.254,Z 844.912,A -85,B 0,C 180,E1 10271.11,E2 10271.11} C_VEL
LIN {X 0,Y 561.692,Z 824.304,A -85,B 0,C 180,E1 10274.05,E2 10274.05} C_VEL
LIN {X 0,Y 563.724,Z 798.21,A -85,B 0,C 180,E1 10276.693,E2 10276.693} C_VEL
LIN {X 0,Y 565.879,Z 767.078,A -85,B 0,C 180,E1 10278.943,E2 10278.943} C_VEL
LIN {X 0,Y 568.098,Z 731.598,A -85,B 0,C 180,E1 10280.744,E2 10280.744} C_VEL
LIN {X 0,Y 570.257,Z 692.379,A -85,B 0,C 180,E1 10282.047,E2 10282.047} C_VEL
LIN {X 0,Y 572.095,Z 642.891,A -85,B 0,C 180,E1 10283.103,E2 10283.103} C_VEL
LIN {X 0,Y 559.722,Z 610.937,A -85,B 0,C 180,E1 10284.741,E2 10284.741} C_VEL
LIN {X 0,Y 555.803,Z 601.31,A -85,B 0,C 180,E1 10285.408,E2 10285.408} C_VEL
LIN {X 0,Y 555.686,Z 601.31,A -85,B 0,C 180,E1 10291.198,E2 10291.198} C_VEL
LIN {X 0,Y 555.571,Z 601.31,A -85,B 0,C 180,E1 10296.863,E2 10296.863} C_VEL
LIN {X 0,Y 555.588,Z 601.31,A -85,B 0,C 180,E1 10302.976,E2 10302.976} C_VEL
LIN {X 0,Y 555.482,Z 601.31,A -85,B 0,C 180,E1 10309.112,E2 10309.112} C_VEL
LIN {X 0,Y 555.492,Z 601.31,A -85,B 0,C 180,E1 10309.647,E2 10309.647} C_VEL
LIN {X 0,Y 570.546,Z 636.401,A -85,B 0,C 180,E1 10311.335,E2 10311.335} C_VEL
LIN {X 0,Y 582.25,Z 668.285,A -85,B 0,C 180,E1 10312.509,E2 10312.509} C_VEL
LIN {X 0,Y 582.85,Z 676.432,A -85,B 0,C 180,E1 10312.655,E2 10312.655} C_VEL
LIN {X 0,Y 575.05,Z 700.26,A -85,B 0,C 180,E1 10312.618,E2 10312.618} C_VEL
LIN {X 0,Y 574.849,Z 702.529,A -85,B 0,C 180,E1 10312.656,E2 10312.656} C_VEL
LIN {X 0,Y 572.343,Z 745.451,A -85,B 0,C 180,E1 10313.752,E2 10313.752} C_VEL
LIN {X 0,Y 569.028,Z 789.201,A -85,B 0,C 180,E1 10315.49,E2 10315.49} C_VEL
LIN {X 0,Y 564.877,Z 832.335,A -85,B 0,C 180,E1 10317.902,E2 10317.902} C_VEL
LIN {X 0,Y 560.615,Z 872.211,A -85,B 0,C 180,E1 10320.894,E2 10320.894} C_VEL
LIN {X 0,Y 556.658,Z 907.938,A -85,B 0,C 180,E1 10324.403,E2 10324.403} C_VEL
LIN {X 0,Y 553.31,Z 939.147,A -85,B 0,C 180,E1 10328.405,E2 10328.405} C_VEL
LIN {X 0,Y 551.123,Z 962.885,A -85,B 0,C 180,E1 10332.401,E2 10332.401} C_VEL
LIN {X 0,Y 549.82,Z 981.072,A -85,B 0,C 180,E1 10336.457,E2 10336.457} C_VEL
LIN {X 0,Y 549.153,Z 994.915,A -85,B 0,C 180,E1 10340.876,E2 10340.876} C_VEL
LIN {X 0,Y 548.95,Z 1003.149,A -85,B 0,C 180,E1 10345.255,E2 10345.255} C_VEL
LIN {X 0,Y 548.959,Z 1005.888,A -85,B 0,C 180,E1 10348.423,E2 10348.423} C_VEL
LIN {X 0,Y 548.825,Z 1005.893,A -85,B 0,C 180,E1 10351.586,E2 10351.586} C_VEL
LIN {X 0,Y 549.018,Z 1000.868,A -85,B 0,C 180,E1 10356.342,E2 10356.342} C_VEL
LIN {X 0,Y 549.331,Z 990.861,A -85,B 0,C 180,E1 10360.735,E2 10360.735} C_VEL
LIN {X 0,Y 550.362,Z 974.724,A -85,B 0,C 180,E1 10365.279,E2 10365.279} C_VEL
LIN {X 0,Y 552.384,Z 951.807,A -85,B 0,C 180,E1 10369.848,E2 10369.848} C_VEL
LIN {X 0,Y 555.28,Z 924.64,A -85,B 0,C 180,E1 10373.921,E2 10373.921} C_VEL
LIN {X 0,Y 558.963,Z 894.455,A -85,B 0,C 180,E1 10377.445,E2 10377.445} C_VEL
LIN {X 0,Y 563.539,Z 858.372,A -85,B 0,C 180,E1 10380.726,E2 10380.726} C_VEL
LIN {X 0,Y 568.264,Z 818.383,A -85,B 0,C 180,E1 10383.497,E2 10383.497} C_VEL
LIN {X 0,Y 572.873,Z 773.35,A -85,B 0,C 180,E1 10385.777,E2 10385.777} C_VEL
LIN {X 0,Y 576.617,Z 727.536,A -85,B 0,C 180,E1 10387.349,E2 10387.349} C_VEL
LIN {X 0,Y 578.72,Z 681.913,A -85,B 0,C 180,E1 10388.283,E2 10388.283} C_VEL
LIN {X 0,Y 578.279,Z 670.025,A -85,B 0,C 180,E1 10388.496,E2 10388.496} C_VEL
LIN {X 0,Y 547.672,Z 601.31,A -85,B 0,C 180,E1 10391.611,E2 10391.611} C_VEL
LIN {X 0,Y 547.583,Z 601.31,A -85,B 0,C 180,E1 10398.347,E2 10398.347} C_VEL
LIN {X 0,Y 547.543,Z 601.31,A -85,B 0,C 180,E1 10404.476,E2 10404.476} C_VEL
LIN {X 0,Y 547.751,Z 601.31,A -85,B 0,C 180,E1 10410.142,E2 10410.142} C_VEL
LIN {X 0,Y 547.951,Z 601.31,A -85,B 0,C 180,E1 10415.867,E2 10415.867} C_VEL
LIN {X 0,Y 548.045,Z 601.31,A -85,B 0,C 180,E1 10420.626,E2 10420.626} C_VEL
LIN {X 0,Y 548.135,Z 601.31,A -85,B 0,C 180,E1 10425.595,E2 10425.595} C_VEL
LIN {X 0,Y 548.327,Z 601.31,A -85,B 0,C 180,E1 10430.456,E2 10430.456} C_VEL
LIN {X 0,Y 548.562,Z 601.31,A -85,B 0,C 180,E1 10435.246,E2 10435.246} C_VEL
LIN {X 0,Y 548.765,Z 601.31,A -85,B 0,C 180,E1 10441.58,E2 10441.58} C_VEL
LIN {X 0,Y 548.521,Z 601.31,A -85,B 0,C 180,E1 10446.34,E2 10446.34} C_VEL
LIN {X 0,Y 548.302,Z 601.31,A -85,B 0,C 180,E1 10451.149,E2 10451.149} C_VEL
LIN {X 0,Y 548.155,Z 601.31,A -85,B 0,C 180,E1 10456.041,E2 10456.041} C_VEL
LIN {X 0,Y 548.023,Z 601.31,A -85,B 0,C 180,E1 10461.058,E2 10461.058} C_VEL
LIN {X 0,Y 547.861,Z 601.31,A -85,B 0,C 180,E1 10466.256,E2 10466.256} C_VEL
LIN {X 0,Y 547.739,Z 601.31,A -85,B 0,C 180,E1 10471.698,E2 10471.698} C_VEL
LIN {X 0,Y 547.605,Z 601.31,A -85,B 0,C 180,E1 10477.486,E2 10477.486} C_VEL
LIN {X 0,Y 547.616,Z 601.31,A -85,B 0,C 180,E1 10483.753,E2 10483.753} C_VEL
LIN {X 0,Y 547.563,Z 601.31,A -85,B 0,C 180,E1 10488.379,E2 10488.379} C_VEL
LIN {X 0,Y 547.554,Z 601.31,A -85,B 0,C 180,E1 10494.466,E2 10494.466} C_VEL
LIN {X 0,Y 547.831,Z 601.423,A -85,B 0,C 180,E1 10498.226,E2 10498.226} C_VEL
LIN {X 0,Y 563.023,Z 642.453,A -85,B 0,C 180,E1 10500.146,E2 10500.146} C_VEL
LIN {X 0,Y 566.643,Z 658.884,A -85,B 0,C 180,E1 10500.882,E2 10500.882} C_VEL
LIN {X 0,Y 564.032,Z 699.089,A -85,B 0,C 180,E1 10502.525,E2 10502.525} C_VEL
LIN {X 0,Y 560.903,Z 735.659,A -85,B 0,C 180,E1 10504.708,E2 10504.708} C_VEL
LIN {X 0,Y 557.58,Z 768.741,A -85,B 0,C 180,E1 10507.393,E2 10507.393} C_VEL
LIN {X 0,Y 554.588,Z 797.891,A -85,B 0,C 180,E1 10510.562,E2 10510.562} C_VEL
LIN {X 0,Y 552.281,Z 821.975,A -85,B 0,C 180,E1 10514.072,E2 10514.072} C_VEL
LIN {X 0,Y 550.713,Z 841.05,A -85,B 0,C 180,E1 10517.871,E2 10517.871} C_VEL
LIN {X 0,Y 549.899,Z 854.26,A -85,B 0,C 180,E1 10521.678,E2 10521.678} C_VEL
LIN {X 0,Y 549.532,Z 861.93,A -85,B 0,C 180,E1 10525.251,E2 10525.251} C_VEL
LIN {X 0,Y 549.349,Z 865.213,A -85,B 0,C 180,E1 10528.415,E2 10528.415} C_VEL
LIN {X 0,Y 549.484,Z 865.143,A -85,B 0,C 180,E1 10531.576,E2 10531.576} C_VEL
LIN {X 0,Y 549.63,Z 860.468,A -85,B 0,C 180,E1 10535.533,E2 10535.533} C_VEL
LIN {X 0,Y 550.038,Z 850.441,A -85,B 0,C 180,E1 10539.509,E2 10539.509} C_VEL
LIN {X 0,Y 551.088,Z 836.334,A -85,B 0,C 180,E1 10543.106,E2 10543.106} C_VEL
LIN {X 0,Y 552.844,Z 815.869,A -85,B 0,C 180,E1 10546.827,E2 10546.827} C_VEL
LIN {X 0,Y 555.408,Z 790.4,A -85,B 0,C 180,E1 10550.246,E2 10550.246} C_VEL
LIN {X 0,Y 558.614,Z 759.254,A -85,B 0,C 180,E1 10553.366,E2 10553.366} C_VEL
LIN {X 0,Y 561.848,Z 725.48,A -85,B 0,C 180,E1 10555.879,E2 10555.879} C_VEL
LIN {X 0,Y 564.687,Z 690.343,A -85,B 0,C 180,E1 10557.796,E2 10557.796} C_VEL
LIN {X 0,Y 566.166,Z 655.264,A -85,B 0,C 180,E1 10559.177,E2 10559.177} C_VEL
LIN {X 0,Y 556.677,Z 623.864,A -85,B 0,C 180,E1 10560.605,E2 10560.605} C_VEL
LIN {X 0,Y 547.754,Z 601.31,A -85,B 0,C 180,E1 10561.702,E2 10561.702} C_VEL
LIN {X 0,Y 547.626,Z 601.31,A -85,B 0,C 180,E1 10567.491,E2 10567.491} C_VEL
LIN {X 0,Y 547.61,Z 601.31,A -85,B 0,C 180,E1 10573.762,E2 10573.762} C_VEL
LIN {X 0,Y 547.559,Z 601.31,A -85,B 0,C 180,E1 10578.398,E2 10578.398} C_VEL
LIN {X 0,Y 547.561,Z 601.31,A -85,B 0,C 180,E1 10584.483,E2 10584.483} C_VEL
LIN {X 0,Y 547.763,Z 601.31,A -85,B 0,C 180,E1 10590.147,E2 10590.147} C_VEL
LIN {X 0,Y 547.961,Z 601.31,A -85,B 0,C 180,E1 10596.041,E2 10596.041} C_VEL
LIN {X 0,Y 561.449,Z 645.354,A -85,B 0,C 180,E1 10597.388,E2 10597.388} C_VEL
LIN {X 0,Y 560.033,Z 696.998,A -85,B 0,C 180,E1 10598.324,E2 10598.324} C_VEL
LIN {X 0,Y 558.299,Z 733.967,A -85,B 0,C 180,E1 10599.606,E2 10599.606} C_VEL
LIN {X 0,Y 556.221,Z 768.063,A -85,B 0,C 180,E1 10601.441,E2 10601.441} C_VEL
LIN {X 0,Y 554.147,Z 798.741,A -85,B 0,C 180,E1 10603.808,E2 10603.808} C_VEL
LIN {X 0,Y 552.537,Z 823.451,A -85,B 0,C 180,E1 10606.436,E2 10606.436} C_VEL
LIN {X 0,Y 551.222,Z 844.483,A -85,B 0,C 180,E1 10609.512,E2 10609.512} C_VEL
LIN {X 0,Y 550.489,Z 860.369,A -85,B 0,C 180,E1 10612.919,E2 10612.919} C_VEL
LIN {X 0,Y 550.142,Z 869.544,A -85,B 0,C 180,E1 10616.055,E2 10616.055} C_VEL
LIN {X 0,Y 550.093,Z 873.27,A -85,B 0,C 180,E1 10618.424,E2 10618.424} C_VEL
LIN {X 0,Y 550.151,Z 874.254,A -85,B 0,C 180,E1 10621.58,E2 10621.58} C_VEL
LIN {X 0,Y 550.657,Z 870.505,A -85,B 0,C 180,E1 10624.736,E2 10624.736} C_VEL
LIN {X 0,Y 551.408,Z 860.82,A -85,B 0,C 180,E1 10628.156,E2 10628.156} C_VEL
LIN {X 0,Y 552.618,Z 846.167,A -85,B 0,C 180,E1 10631.265,E2 10631.265} C_VEL
LIN {X 0,Y 554.157,Z 825.658,A -85,B 0,C 180,E1 10634.245,E2 10634.245} C_VEL
LIN {X 0,Y 556.303,Z 799.64,A -85,B 0,C 180,E1 10636.922,E2 10636.922} C_VEL
LIN {X 0,Y 558.576,Z 768.709,A -85,B 0,C 180,E1 10639.2,E2 10639.2} C_VEL
LIN {X 0,Y 561.013,Z 732.087,A -85,B 0,C 180,E1 10641.096,E2 10641.096} C_VEL
LIN {X 0,Y 563.418,Z 691.569,A -85,B 0,C 180,E1 10642.464,E2 10642.464} C_VEL
LIN {X 0,Y 565.249,Z 644.709,A -85,B 0,C 180,E1 10643.497,E2 10643.497} C_VEL
LIN {X 0,Y 553.615,Z 614.711,A -85,B 0,C 180,E1 10645.12,E2 10645.12} C_VEL
LIN {X 0,Y 547.85,Z 601.31,A -85,B 0,C 180,E1 10646.044,E2 10646.044} C_VEL
LIN {X 0,Y 547.782,Z 601.31,A -85,B 0,C 180,E1 10651.7,E2 10651.7} C_VEL
LIN {X 0,Y 547.659,Z 601.31,A -85,B 0,C 180,E1 10657.487,E2 10657.487} C_VEL
LIN {X 0,Y 547.618,Z 601.31,A -85,B 0,C 180,E1 10663.758,E2 10663.758} C_VEL
LIN {X 0,Y 547.569,Z 601.312,A -85,B 0,C 180,E1 10668.98,E2 10668.98} C_VEL
LIN {X 0,Y 553.678,Z 614.672,A -85,B 0,C 180,E1 10669.751,E2 10669.751} C_VEL
LIN {X 0,Y 565.201,Z 642.108,A -85,B 0,C 180,E1 10671.06,E2 10671.06} C_VEL
LIN {X 0,Y 575.553,Z 671.033,A -85,B 0,C 180,E1 10672.152,E2 10672.152} C_VEL
LIN {X 0,Y 574.849,Z 702.529,A -85,B 0,C 180,E1 10672.656,E2 10672.656} C_VEL
LIN {X 0,Y 570.445,Z 719.458,A -85,B 0,C 180,E1 10672.818,E2 10672.818} C_VEL
LIN {X 0,Y 566.155,Z 734.083,A -85,B 0,C 180,E1 10673.013,E2 10673.013} C_VEL
LIN {X 0,Y 565.986,Z 736.189,A -85,B 0,C 180,E1 10673.073,E2 10673.073} C_VEL
LIN {X 0,Y 562.609,Z 779.896,A -85,B 0,C 180,E1 10674.701,E2 10674.701} C_VEL
LIN {X 0,Y 558.598,Z 821.796,A -85,B 0,C 180,E1 10676.919,E2 10676.919} C_VEL
LIN {X 0,Y 554.374,Z 860.629,A -85,B 0,C 180,E1 10679.668,E2 10679.668} C_VEL
LIN {X 0,Y 550.309,Z 896.049,A -85,B 0,C 180,E1 10682.917,E2 10682.917} C_VEL
LIN {X 0,Y 546.59,Z 929.127,A -85,B 0,C 180,E1 10686.862,E2 10686.862} C_VEL
LIN {X 0,Y 543.79,Z 956.629,A -85,B 0,C 180,E1 10691.186,E2 10691.186} C_VEL
LIN {X 0,Y 542.206,Z 976.726,A -85,B 0,C 180,E1 10695.438,E2 10695.438} C_VEL
LIN {X 0,Y 541.442,Z 990.763,A -85,B 0,C 180,E1 10699.524,E2 10699.524} C_VEL
LIN {X 0,Y 541.138,Z 999.84,A -85,B 0,C 180,E1 10703.574,E2 10703.574} C_VEL
LIN {X 0,Y 541.099,Z 1005.018,A -85,B 0,C 180,E1 10708.4,E2 10708.4} C_VEL
LIN {X 0,Y 540.968,Z 1005.044,A -85,B 0,C 180,E1 10711.609,E2 10711.609} C_VEL
LIN {X 0,Y 541.16,Z 1001.32,A -85,B 0,C 180,E1 10715.62,E2 10715.62} C_VEL
LIN {X 0,Y 541.415,Z 991.168,A -85,B 0,C 180,E1 10720.485,E2 10720.485} C_VEL
LIN {X 0,Y 542.426,Z 975.279,A -85,B 0,C 180,E1 10725.133,E2 10725.133} C_VEL
LIN {X 0,Y 544.299,Z 954.246,A -85,B 0,C 180,E1 10729.52,E2 10729.52} C_VEL
LIN {X 0,Y 547.142,Z 928.39,A -85,B 0,C 180,E1 10733.612,E2 10733.612} C_VEL
LIN {X 0,Y 551.136,Z 897.267,A -85,B 0,C 180,E1 10737.412,E2 10737.412} C_VEL
LIN {X 0,Y 556.023,Z 859.458,A -85,B 0,C 180,E1 10740.948,E2 10740.948} C_VEL
LIN {X 0,Y 560.993,Z 819.266,A -85,B 0,C 180,E1 10743.788,E2 10743.788} C_VEL
LIN {X 0,Y 565.758,Z 774.37,A -85,B 0,C 180,E1 10746.106,E2 10746.106} C_VEL
LIN {X 0,Y 569.74,Z 726.882,A -85,B 0,C 180,E1 10747.757,E2 10747.757} C_VEL
LIN {X 0,Y 572.013,Z 680.073,A -85,B 0,C 180,E1 10748.713,E2 10748.713} C_VEL
LIN {X 0,Y 571.228,Z 671.878,A -85,B 0,C 180,E1 10748.889,E2 10748.889} C_VEL
LIN {X 0,Y 539.692,Z 601.31,A -85,B 0,C 180,E1 10752.117,E2 10752.117} C_VEL
LIN {X 0,Y 539.61,Z 601.31,A -85,B 0,C 180,E1 10757.639,E2 10757.639} C_VEL
LIN {X 0,Y 539.617,Z 601.31,A -85,B 0,C 180,E1 10763.873,E2 10763.873} C_VEL
LIN {X 0,Y 539.843,Z 601.31,A -85,B 0,C 180,E1 10769.659,E2 10769.659} C_VEL
LIN {X 0,Y 539.965,Z 601.31,A -85,B 0,C 180,E1 10775.111,E2 10775.111} C_VEL
LIN {X 0,Y 540.127,Z 601.31,A -85,B 0,C 180,E1 10780.33,E2 10780.33} C_VEL
LIN {X 0,Y 540.227,Z 601.31,A -85,B 0,C 180,E1 10785.38,E2 10785.38} C_VEL
LIN {X 0,Y 540.405,Z 601.31,A -85,B 0,C 180,E1 10790.315,E2 10790.315} C_VEL
LIN {X 0,Y 540.662,Z 601.31,A -85,B 0,C 180,E1 10795.176,E2 10795.176} C_VEL
LIN {X 0,Y 540.796,Z 601.31,A -85,B 0,C 180,E1 10799.998,E2 10799.998} C_VEL
LIN {X 0,Y 540.705,Z 601.31,A -85,B 0,C 180,E1 10804.819,E2 10804.819} C_VEL
LIN {X 0,Y 540.399,Z 601.31,A -85,B 0,C 180,E1 10811.314,E2 10811.314} C_VEL
LIN {X 0,Y 540.219,Z 601.31,A -85,B 0,C 180,E1 10817.502,E2 10817.502} C_VEL
LIN {X 0,Y 540.053,Z 601.31,A -85,B 0,C 180,E1 10823.121,E2 10823.121} C_VEL
LIN {X 0,Y 539.86,Z 601.31,A -85,B 0,C 180,E1 10828.489,E2 10828.489} C_VEL
LIN {X 0,Y 539.717,Z 601.31,A -85,B 0,C 180,E1 10834.148,E2 10834.148} C_VEL
LIN {X 0,Y 539.628,Z 601.31,A -85,B 0,C 180,E1 10840.213,E2 10840.213} C_VEL
LIN {X 0,Y 539.642,Z 601.31,A -85,B 0,C 180,E1 10845.41,E2 10845.41} C_VEL
LIN {X 0,Y 539.606,Z 601.31,A -85,B 0,C 180,E1 10851.842,E2 10851.842} C_VEL
LIN {X 0,Y 539.909,Z 601.904,A -85,B 0,C 180,E1 10857.707,E2 10857.707} C_VEL
LIN {X 0,Y 555.781,Z 643.131,A -85,B 0,C 180,E1 10859.731,E2 10859.731} C_VEL
LIN {X 0,Y 559.647,Z 661.14,A -85,B 0,C 180,E1 10860.554,E2 10860.554} C_VEL
LIN {X 0,Y 556.97,Z 700.765,A -85,B 0,C 180,E1 10862.208,E2 10862.208} C_VEL
LIN {X 0,Y 553.769,Z 736.372,A -85,B 0,C 180,E1 10864.361,E2 10864.361} C_VEL
LIN {X 0,Y 550.362,Z 769.068,A -85,B 0,C 180,E1 10867.039,E2 10867.039} C_VEL
LIN {X 0,Y 547.169,Z 798.578,A -85,B 0,C 180,E1 10870.268,E2 10870.268} C_VEL
LIN {X 0,Y 544.651,Z 822.843,A -85,B 0,C 180,E1 10873.843,E2 10873.843} C_VEL
LIN {X 0,Y 542.985,Z 842.105,A -85,B 0,C 180,E1 10877.733,E2 10877.733} C_VEL
LIN {X 0,Y 542.116,Z 855.198,A -85,B 0,C 180,E1 10881.558,E2 10881.558} C_VEL
LIN {X 0,Y 541.712,Z 862.902,A -85,B 0,C 180,E1 10885.182,E2 10885.182} C_VEL
LIN {X 0,Y 541.523,Z 866.196,A -85,B 0,C 180,E1 10888.392,E2 10888.392} C_VEL
LIN {X 0,Y 541.672,Z 866.126,A -85,B 0,C 180,E1 10891.599,E2 10891.599} C_VEL
LIN {X 0,Y 541.83,Z 861.43,A -85,B 0,C 180,E1 10895.612,E2 10895.612} C_VEL
LIN {X 0,Y 542.267,Z 851.372,A -85,B 0,C 180,E1 10899.647,E2 10899.647} C_VEL
LIN {X 0,Y 543.394,Z 837.228,A -85,B 0,C 180,E1 10903.295,E2 10903.295} C_VEL
LIN {X 0,Y 545.16,Z 817.917,A -85,B 0,C 180,E1 10906.879,E2 10906.879} C_VEL
LIN {X 0,Y 547.729,Z 793.28,A -85,B 0,C 180,E1 10910.285,E2 10910.285} C_VEL
LIN {X 0,Y 551.084,Z 762.366,A -85,B 0,C 180,E1 10913.491,E2 10913.491} C_VEL
LIN {X 0,Y 554.64,Z 727.71,A -85,B 0,C 180,E1 10916.132,E2 10916.132} C_VEL
LIN {X 0,Y 557.648,Z 691.792,A -85,B 0,C 180,E1 10918.131,E2 10918.131} C_VEL
LIN {X 0,Y 559.193,Z 657.376,A -85,B 0,C 180,E1 10919.513,E2 10919.513} C_VEL
LIN {X 0,Y 550.509,Z 627.974,A -85,B 0,C 180,E1 10920.888,E2 10920.888} C_VEL
LIN {X 0,Y 539.773,Z 601.31,A -85,B 0,C 180,E1 10922.227,E2 10922.227} C_VEL
LIN {X 0,Y 539.687,Z 601.31,A -85,B 0,C 180,E1 10928.195,E2 10928.195} C_VEL
LIN {X 0,Y 539.669,Z 601.31,A -85,B 0,C 180,E1 10934.574,E2 10934.574} C_VEL
LIN {X 0,Y 539.597,Z 601.31,A -85,B 0,C 180,E1 10939.784,E2 10939.784} C_VEL
LIN {X 0,Y 539.688,Z 601.31,A -85,B 0,C 180,E1 10945.85,E2 10945.85} C_VEL
LIN {X 0,Y 539.868,Z 601.31,A -85,B 0,C 180,E1 10951.511,E2 10951.511} C_VEL
LIN {X 0,Y 540.035,Z 601.31,A -85,B 0,C 180,E1 10955.664,E2 10955.664} C_VEL
LIN {X 0,Y 554.126,Z 646.514,A -85,B 0,C 180,E1 10957.101,E2 10957.101} C_VEL
LIN {X 0,Y 552.546,Z 698.933,A -85,B 0,C 180,E1 10958.089,E2 10958.089} C_VEL
LIN {X 0,Y 550.778,Z 735.321,A -85,B 0,C 180,E1 10959.397,E2 10959.397} C_VEL
LIN {X 0,Y 548.571,Z 769.468,A -85,B 0,C 180,E1 10961.277,E2 10961.277} C_VEL
LIN {X 0,Y 546.502,Z 799.421,A -85,B 0,C 180,E1 10963.626,E2 10963.626} C_VEL
LIN {X 0,Y 544.677,Z 826.032,A -85,B 0,C 180,E1 10966.521,E2 10966.521} C_VEL
LIN {X 0,Y 543.311,Z 847.246,A -85,B 0,C 180,E1 10969.763,E2 10969.763} C_VEL
LIN {X 0,Y 542.672,Z 861.667,A -85,B 0,C 180,E1 10972.963,E2 10972.963} C_VEL
LIN {X 0,Y 542.318,Z 870.438,A -85,B 0,C 180,E1 10975.998,E2 10975.998} C_VEL
LIN {X 0,Y 542.274,Z 874.264,A -85,B 0,C 180,E1 10978.401,E2 10978.401} C_VEL
LIN {X 0,Y 542.352,Z 875.343,A -85,B 0,C 180,E1 10981.603,E2 10981.603} C_VEL
LIN {X 0,Y 542.869,Z 871.69,A -85,B 0,C 180,E1 10984.804,E2 10984.804} C_VEL
LIN {X 0,Y 543.711,Z 861.852,A -85,B 0,C 180,E1 10988.332,E2 10988.332} C_VEL
LIN {X 0,Y 545.086,Z 846.386,A -85,B 0,C 180,E1 10991.626,E2 10991.626} C_VEL
LIN {X 0,Y 546.797,Z 825.365,A -85,B 0,C 180,E1 10994.646,E2 10994.646} C_VEL
LIN {X 0,Y 549.107,Z 798.826,A -85,B 0,C 180,E1 10997.357,E2 10997.357} C_VEL
LIN {X 0,Y 551.521,Z 767.379,A -85,B 0,C 180,E1 10999.664,E2 10999.664} C_VEL
LIN {X 0,Y 554.162,Z 730.597,A -85,B 0,C 180,E1 11001.552,E2 11001.552} C_VEL
LIN {X 0,Y 556.768,Z 689.112,A -85,B 0,C 180,E1 11002.94,E2 11002.94} C_VEL
LIN {X 0,Y 558.46,Z 646.616,A -85,B 0,C 180,E1 11003.905,E2 11003.905} C_VEL
LIN {X 0,Y 546.752,Z 616.334,A -85,B 0,C 180,E1 11005.637,E2 11005.637} C_VEL
LIN {X 0,Y 539.903,Z 601.31,A -85,B 0,C 180,E1 11006.768,E2 11006.768} C_VEL
LIN {X 0,Y 539.776,Z 601.31,A -85,B 0,C 180,E1 11012.643,E2 11012.643} C_VEL
LIN {X 0,Y 539.71,Z 601.31,A -85,B 0,C 180,E1 11018.186,E2 11018.186} C_VEL
LIN {X 0,Y 539.651,Z 601.31,A -85,B 0,C 180,E1 11024.573,E2 11024.573} C_VEL
LIN {X 0,Y 539.646,Z 601.31,A -85,B 0,C 180,E1 11028.207,E2 11028.207} C_VEL
LIN {X 0,Y 544.564,Z 611.788,A -85,B 0,C 180,E1 11028.915,E2 11028.915} C_VEL
LIN {X 0,Y 557.192,Z 639.834,A -85,B 0,C 180,E1 11030.45,E2 11030.45} C_VEL
LIN {X 0,Y 568.813,Z 674.628,A -85,B 0,C 180,E1 11031.785,E2 11031.785} C_VEL
LIN {X 0,Y 566.92,Z 723.267,A -85,B 0,C 180,E1 11032.713,E2 11032.713} C_VEL
LIN {X 0,Y 565.986,Z 736.189,A -85,B 0,C 180,E1 11033.073,E2 11033.073} C_VEL
LIN {X 0,Y 561.346,Z 752.785,A -85,B 0,C 180,E1 11033.415,E2 11033.415} C_VEL
LIN {X 0,Y 556.838,Z 767.083,A -85,B 0,C 180,E1 11033.772,E2 11033.772} C_VEL
LIN {X 0,Y 556.623,Z 769.115,A -85,B 0,C 180,E1 11033.851,E2 11033.851} C_VEL
LIN {X 0,Y 552.569,Z 811.736,A -85,B 0,C 180,E1 11035.976,E2 11035.976} C_VEL
LIN {X 0,Y 548.226,Z 850.259,A -85,B 0,C 180,E1 11038.562,E2 11038.562} C_VEL
LIN {X 0,Y 544.058,Z 885.051,A -85,B 0,C 180,E1 11041.577,E2 11041.577} C_VEL
LIN {X 0,Y 540.009,Z 918.207,A -85,B 0,C 180,E1 11045.268,E2 11045.268} C_VEL
LIN {X 0,Y 536.785,Z 947.695,A -85,B 0,C 180,E1 11049.559,E2 11049.559} C_VEL
LIN {X 0,Y 534.814,Z 970.749,A -85,B 0,C 180,E1 11054.054,E2 11054.054} C_VEL
LIN {X 0,Y 533.747,Z 987.271,A -85,B 0,C 180,E1 11058.543,E2 11058.543} C_VEL
LIN {X 0,Y 533.306,Z 997.468,A -85,B 0,C 180,E1 11062.659,E2 11062.659} C_VEL
LIN {X 0,Y 533.17,Z 1003.075,A -85,B 0,C 180,E1 11066.746,E2 11066.746} C_VEL
LIN {X 0,Y 533.222,Z 1004.537,A -85,B 0,C 180,E1 11070.004,E2 11070.004} C_VEL
LIN {X 0,Y 533.265,Z 1001.528,A -85,B 0,C 180,E1 11074.894,E2 11074.894} C_VEL
LIN {X 0,Y 533.427,Z 993.38,A -85,B 0,C 180,E1 11079.405,E2 11079.405} C_VEL
LIN {X 0,Y 534.138,Z 979.77,A -85,B 0,C 180,E1 11083.957,E2 11083.957} C_VEL
LIN {X 0,Y 535.687,Z 960.914,A -85,B 0,C 180,E1 11088.342,E2 11088.342} C_VEL
LIN {X 0,Y 538.281,Z 937.26,A -85,B 0,C 180,E1 11092.492,E2 11092.492} C_VEL
LIN {X 0,Y 542.254,Z 906.999,A -85,B 0,C 180,E1 11096.562,E2 11096.562} C_VEL
LIN {X 0,Y 547.081,Z 871.453,A -85,B 0,C 180,E1 11100.219,E2 11100.219} C_VEL
LIN {X 0,Y 552.199,Z 832.3,A -85,B 0,C 180,E1 11103.289,E2 11103.289} C_VEL
LIN {X 0,Y 557.302,Z 789.129,A -85,B 0,C 180,E1 11105.793,E2 11105.793} C_VEL
LIN {X 0,Y 561.618,Z 744.278,A -85,B 0,C 180,E1 11107.622,E2 11107.622} C_VEL
LIN {X 0,Y 564.531,Z 697.801,A -85,B 0,C 180,E1 11108.825,E2 11108.825} C_VEL
LIN {X 0,Y 564.737,Z 674.957,A -85,B 0,C 180,E1 11109.232,E2 11109.232} C_VEL
LIN {X 0,Y 531.739,Z 601.31,A -85,B 0,C 180,E1 11112.711,E2 11112.711} C_VEL
LIN {X 0,Y 531.688,Z 601.31,A -85,B 0,C 180,E1 11119.054,E2 11119.054} C_VEL
LIN {X 0,Y 531.723,Z 601.31,A -85,B 0,C 180,E1 11125.261,E2 11125.261} C_VEL
LIN {X 0,Y 531.937,Z 601.31,A -85,B 0,C 180,E1 11131.042,E2 11131.042} C_VEL
LIN {X 0,Y 532.096,Z 601.31,A -85,B 0,C 180,E1 11136.508,E2 11136.508} C_VEL
LIN {X 0,Y 532.237,Z 601.31,A -85,B 0,C 180,E1 11141.752,E2 11141.752} C_VEL
LIN {X 0,Y 532.334,Z 601.31,A -85,B 0,C 180,E1 11146.839,E2 11146.839} C_VEL
LIN {X 0,Y 532.627,Z 601.31,A -85,B 0,C 180,E1 11151.822,E2 11151.822} C_VEL
LIN {X 0,Y 532.821,Z 601.31,A -85,B 0,C 180,E1 11156.738,E2 11156.738} C_VEL
LIN {X 0,Y 532.956,Z 601.31,A -85,B 0,C 180,E1 11161.627,E2 11161.627} C_VEL
LIN {X 0,Y 532.682,Z 601.31,A -85,B 0,C 180,E1 11166.53,E2 11166.53} C_VEL
LIN {X 0,Y 532.47,Z 601.31,A -85,B 0,C 180,E1 11171.485,E2 11171.485} C_VEL
LIN {X 0,Y 532.332,Z 601.31,A -85,B 0,C 180,E1 11176.531,E2 11176.531} C_VEL
LIN {X 0,Y 532.166,Z 601.31,A -85,B 0,C 180,E1 11181.717,E2 11181.717} C_VEL
LIN {X 0,Y 531.928,Z 601.31,A -85,B 0,C 180,E1 11187.979,E2 11187.979} C_VEL
LIN {X 0,Y 531.802,Z 601.31,A -85,B 0,C 180,E1 11194.275,E2 11194.275} C_VEL
LIN {X 0,Y 531.675,Z 601.31,A -85,B 0,C 180,E1 11199.687,E2 11199.687} C_VEL
LIN {X 0,Y 531.741,Z 601.31,A -85,B 0,C 180,E1 11205.413,E2 11205.413} C_VEL
LIN {X 0,Y 531.651,Z 601.31,A -85,B 0,C 180,E1 11211.165,E2 11211.165} C_VEL
LIN {X 0,Y 531.928,Z 601.31,A -85,B 0,C 180,E1 11217.117,E2 11217.117} C_VEL
LIN {X 0,Y 549.326,Z 646.742,A -85,B 0,C 180,E1 11219.443,E2 11219.443} C_VEL
LIN {X 0,Y 552.712,Z 662.936,A -85,B 0,C 180,E1 11220.201,E2 11220.201} C_VEL
LIN {X 0,Y 549.831,Z 703.208,A -85,B 0,C 180,E1 11221.922,E2 11221.922} C_VEL
LIN {X 0,Y 546.53,Z 738.321,A -85,B 0,C 180,E1 11224.091,E2 11224.091} C_VEL
LIN {X 0,Y 542.884,Z 771.668,A -85,B 0,C 180,E1 11226.886,E2 11226.886} C_VEL
LIN {X 0,Y 539.575,Z 800.605,A -85,B 0,C 180,E1 11230.14,E2 11230.14} C_VEL
LIN {X 0,Y 536.98,Z 824.44,A -85,B 0,C 180,E1 11233.733,E2 11233.733} C_VEL
LIN {X 0,Y 535.27,Z 843.024,A -85,B 0,C 180,E1 11237.553,E2 11237.553} C_VEL
LIN {X 0,Y 534.329,Z 856.148,A -85,B 0,C 180,E1 11241.434,E2 11241.434} C_VEL
LIN {X 0,Y 533.895,Z 863.876,A -85,B 0,C 180,E1 11245.111,E2 11245.111} C_VEL
LIN {X 0,Y 533.702,Z 867.18,A -85,B 0,C 180,E1 11248.369,E2 11248.369} C_VEL
LIN {X 0,Y 533.848,Z 867.11,A -85,B 0,C 180,E1 11251.622,E2 11251.622} C_VEL
LIN {X 0,Y 534.034,Z 862.396,A -85,B 0,C 180,E1 11255.695,E2 11255.695} C_VEL
LIN {X 0,Y 534.496,Z 852.315,A -85,B 0,C 180,E1 11259.788,E2 11259.788} C_VEL
LIN {X 0,Y 535.723,Z 838.136,A -85,B 0,C 180,E1 11263.489,E2 11263.489} C_VEL
LIN {X 0,Y 537.658,Z 818.277,A -85,B 0,C 180,E1 11267.206,E2 11267.206} C_VEL
LIN {X 0,Y 540.509,Z 792.909,A -85,B 0,C 180,E1 11270.722,E2 11270.722} C_VEL
LIN {X 0,Y 544.041,Z 761.935,A -85,B 0,C 180,E1 11273.923,E2 11273.923} C_VEL
LIN {X 0,Y 547.567,Z 728.408,A -85,B 0,C 180,E1 11276.496,E2 11276.496} C_VEL
LIN {X 0,Y 550.694,Z 692.732,A -85,B 0,C 180,E1 11278.501,E2 11278.501} C_VEL
LIN {X 0,Y 552.189,Z 659.265,A -85,B 0,C 180,E1 11279.87,E2 11279.87} C_VEL
LIN {X 0,Y 544.084,Z 631.384,A -85,B 0,C 180,E1 11281.212,E2 11281.212} C_VEL
LIN {X 0,Y 531.865,Z 601.31,A -85,B 0,C 180,E1 11282.82,E2 11282.82} C_VEL
LIN {X 0,Y 531.721,Z 601.31,A -85,B 0,C 180,E1 11288.817,E2 11288.817} C_VEL
LIN {X 0,Y 531.768,Z 601.31,A -85,B 0,C 180,E1 11294.59,E2 11294.59} C_VEL
LIN {X 0,Y 531.643,Z 601.31,A -85,B 0,C 180,E1 11300.303,E2 11300.303} C_VEL
LIN {X 0,Y 531.774,Z 601.31,A -85,B 0,C 180,E1 11305.713,E2 11305.713} C_VEL
LIN {X 0,Y 531.938,Z 601.31,A -85,B 0,C 180,E1 11311.999,E2 11311.999} C_VEL
LIN {X 0,Y 532.103,Z 601.31,A -85,B 0,C 180,E1 11315.316,E2 11315.316} C_VEL
LIN {X 0,Y 546.744,Z 648.182,A -85,B 0,C 180,E1 11316.829,E2 11316.829} C_VEL
LIN {X 0,Y 545.144,Z 698.936,A -85,B 0,C 180,E1 11317.808,E2 11317.808} C_VEL
LIN {X 0,Y 543.243,Z 736.503,A -85,B 0,C 180,E1 11319.183,E2 11319.183} C_VEL
LIN {X 0,Y 540.931,Z 770.745,A -85,B 0,C 180,E1 11321.109,E2 11321.109} C_VEL
LIN {X 0,Y 538.742,Z 801.268,A -85,B 0,C 180,E1 11323.551,E2 11323.551} C_VEL
LIN {X 0,Y 536.92,Z 827.062,A -85,B 0,C 180,E1 11326.414,E2 11326.414} C_VEL
LIN {X 0,Y 535.543,Z 847.819,A -85,B 0,C 180,E1 11329.613,E2 11329.613} C_VEL
LIN {X 0,Y 534.788,Z 863.391,A -85,B 0,C 180,E1 11333.132,E2 11333.132} C_VEL
LIN {X 0,Y 534.524,Z 872.916,A -85,B 0,C 180,E1 11336.753,E2 11336.753} C_VEL
LIN {X 0,Y 534.485,Z 876.472,A -85,B 0,C 180,E1 11340.002,E2 11340.002} C_VEL
LIN {X 0,Y 534.704,Z 875.316,A -85,B 0,C 180,E1 11343.25,E2 11343.25} C_VEL
LIN {X 0,Y 535.513,Z 868.136,A -85,B 0,C 180,E1 11346.907,E2 11346.907} C_VEL
LIN {X 0,Y 536.715,Z 856.114,A -85,B 0,C 180,E1 11350.163,E2 11350.163} C_VEL
LIN {X 0,Y 538.301,Z 837.667,A -85,B 0,C 180,E1 11353.404,E2 11353.404} C_VEL
LIN {X 0,Y 540.532,Z 814.211,A -85,B 0,C 180,E1 11356.278,E2 11356.278} C_VEL
LIN {X 0,Y 542.999,Z 785.308,A -85,B 0,C 180,E1 11358.834,E2 11358.834} C_VEL
LIN {X 0,Y 545.685,Z 751.929,A -85,B 0,C 180,E1 11360.944,E2 11360.944} C_VEL
LIN {X 0,Y 548.524,Z 713.002,A -85,B 0,C 180,E1 11362.645,E2 11362.645} C_VEL
LIN {X 0,Y 551.443,Z 665.885,A -85,B 0,C 180,E1 11363.912,E2 11363.912} C_VEL
LIN {X 0,Y 551.84,Z 648.588,A -85,B 0,C 180,E1 11364.333,E2 11364.333} C_VEL
LIN {X 0,Y 540.938,Z 620.422,A -85,B 0,C 180,E1 11366.029,E2 11366.029} C_VEL
LIN {X 0,Y 532.021,Z 601.31,A -85,B 0,C 180,E1 11367.675,E2 11367.675} C_VEL
LIN {X 0,Y 531.866,Z 601.31,A -85,B 0,C 180,E1 11372.765,E2 11372.765} C_VEL
LIN {X 0,Y 531.747,Z 601.31,A -85,B 0,C 180,E1 11378.814,E2 11378.814} C_VEL
LIN {X 0,Y 531.751,Z 601.31,A -85,B 0,C 180,E1 11384.579,E2 11384.579} C_VEL
LIN {X 0,Y 531.703,Z 601.31,A -85,B 0,C 180,E1 11387.387,E2 11387.387} C_VEL
LIN {X 0,Y 534.172,Z 607.039,A -85,B 0,C 180,E1 11387.796,E2 11387.796} C_VEL
LIN {X 0,Y 547.27,Z 633.26,A -85,B 0,C 180,E1 11389.553,E2 11389.553} C_VEL
LIN {X 0,Y 562.085,Z 675.769,A -85,B 0,C 180,E1 11391.361,E2 11391.361} C_VEL
LIN {X 0,Y 560.082,Z 724.301,A -85,B 0,C 180,E1 11392.324,E2 11392.324} C_VEL
LIN {X 0,Y 556.623,Z 769.115,A -85,B 0,C 180,E1 11393.851,E2 11393.851} C_VEL
LIN {X 0,Y 551.77,Z 785.214,A -85,B 0,C 180,E1 11394.368,E2 11394.368} C_VEL
LIN {X 0,Y 546.912,Z 798.936,A -85,B 0,C 180,E1 11394.885,E2 11394.885} C_VEL
LIN {X 0,Y 546.632,Z 800.872,A -85,B 0,C 180,E1 11394.989,E2 11394.989} C_VEL
LIN {X 0,Y 541.8,Z 842.076,A -85,B 0,C 180,E1 11397.61,E2 11397.61} C_VEL
LIN {X 0,Y 536.807,Z 882.208,A -85,B 0,C 180,E1 11401.029,E2 11401.029} C_VEL
LIN {X 0,Y 532.483,Z 916.637,A -85,B 0,C 180,E1 11404.88,E2 11404.88} C_VEL
LIN {X 0,Y 529.054,Z 946.501,A -85,B 0,C 180,E1 11409.268,E2 11409.268} C_VEL
LIN {X 0,Y 526.984,Z 969.3,A -85,B 0,C 180,E1 11413.75,E2 11413.75} C_VEL
LIN {X 0,Y 525.912,Z 986.172,A -85,B 0,C 180,E1 11418.35,E2 11418.35} C_VEL
LIN {X 0,Y 525.441,Z 996.521,A -85,B 0,C 180,E1 11422.549,E2 11422.549} C_VEL
LIN {X 0,Y 525.319,Z 1002.19,A -85,B 0,C 180,E1 11426.698,E2 11426.698} C_VEL
LIN {X 0,Y 525.368,Z 1003.68,A -85,B 0,C 180,E1 11430.005,E2 11430.005} C_VEL
LIN {X 0,Y 525.396,Z 1000.683,A -85,B 0,C 180,E1 11434.968,E2 11434.968} C_VEL
LIN {X 0,Y 525.563,Z 992.506,A -85,B 0,C 180,E1 11439.547,E2 11439.547} C_VEL
LIN {X 0,Y 526.309,Z 978.865,A -85,B 0,C 180,E1 11444.169,E2 11444.169} C_VEL
LIN {X 0,Y 527.973,Z 959.259,A -85,B 0,C 180,E1 11448.758,E2 11448.758} C_VEL
LIN {X 0,Y 530.742,Z 935.708,A -85,B 0,C 180,E1 11452.896,E2 11452.896} C_VEL
LIN {X 0,Y 534.55,Z 907.562,A -85,B 0,C 180,E1 11456.734,E2 11456.734} C_VEL
LIN {X 0,Y 539.576,Z 871.555,A -85,B 0,C 180,E1 11460.51,E2 11460.51} C_VEL
LIN {X 0,Y 544.986,Z 831.857,A -85,B 0,C 180,E1 11463.658,E2 11463.658} C_VEL
LIN {X 0,Y 550.281,Z 788.744,A -85,B 0,C 180,E1 11466.183,E2 11466.183} C_VEL
LIN {X 0,Y 554.671,Z 744.257,A -85,B 0,C 180,E1 11468.014,E2 11468.014} C_VEL
LIN {X 0,Y 557.725,Z 697.665,A -85,B 0,C 180,E1 11469.235,E2 11469.235} C_VEL
LIN {X 0,Y 557.788,Z 676.919,A -85,B 0,C 180,E1 11469.625,E2 11469.625} C_VEL
LIN {X 0,Y 523.854,Z 601.31,A -85,B 0,C 180,E1 11473.2,E2 11473.2} C_VEL
LIN {X 0,Y 523.787,Z 601.31,A -85,B 0,C 180,E1 11478.782,E2 11478.782} C_VEL
LIN {X 0,Y 523.731,Z 601.31,A -85,B 0,C 180,E1 11484.653,E2 11484.653} C_VEL
LIN {X 0,Y 523.962,Z 601.31,A -85,B 0,C 180,E1 11490.558,E2 11490.558} C_VEL
LIN {X 0,Y 524.172,Z 601.31,A -85,B 0,C 180,E1 11496.131,E2 11496.131} C_VEL
LIN {X 0,Y 524.295,Z 601.31,A -85,B 0,C 180,E1 11501.466,E2 11501.466} C_VEL
LIN {X 0,Y 524.417,Z 601.31,A -85,B 0,C 180,E1 11506.636,E2 11506.636} C_VEL
LIN {X 0,Y 524.7,Z 601.31,A -85,B 0,C 180,E1 11511.698,E2 11511.698} C_VEL
LIN {X 0,Y 524.929,Z 601.31,A -85,B 0,C 180,E1 11516.689,E2 11516.689} C_VEL
LIN {X 0,Y 525.049,Z 601.31,A -85,B 0,C 180,E1 11521.651,E2 11521.651} C_VEL
LIN {X 0,Y 524.764,Z 601.31,A -85,B 0,C 180,E1 11526.629,E2 11526.629} C_VEL
LIN {X 0,Y 524.551,Z 601.31,A -85,B 0,C 180,E1 11531.661,E2 11531.661} C_VEL
LIN {X 0,Y 524.36,Z 601.31,A -85,B 0,C 180,E1 11537.512,E2 11537.512} C_VEL
LIN {X 0,Y 524.196,Z 601.31,A -85,B 0,C 180,E1 11542.324,E2 11542.324} C_VEL
LIN {X 0,Y 524.051,Z 601.31,A -85,B 0,C 180,E1 11547.547,E2 11547.547} C_VEL
LIN {X 0,Y 523.886,Z 601.31,A -85,B 0,C 180,E1 11553.324,E2 11553.324} C_VEL
LIN {X 0,Y 523.772,Z 601.31,A -85,B 0,C 180,E1 11559.513,E2 11559.513} C_VEL
LIN {X 0,Y 523.83,Z 601.31,A -85,B 0,C 180,E1 11563.95,E2 11563.95} C_VEL
LIN {X 0,Y 523.771,Z 601.31,A -85,B 0,C 180,E1 11568.76,E2 11568.76} C_VEL
LIN {X 0,Y 523.758,Z 601.31,A -85,B 0,C 180,E1 11574.643,E2 11574.643} C_VEL
LIN {X 0,Y 523.931,Z 601.31,A -85,B 0,C 180,E1 11576.554,E2 11576.554} C_VEL
LIN {X 0,Y 542.203,Z 647.76,A -85,B 0,C 180,E1 11579.021,E2 11579.021} C_VEL
LIN {X 0,Y 545.791,Z 664.815,A -85,B 0,C 180,E1 11579.841,E2 11579.841} C_VEL
LIN {X 0,Y 542.791,Z 705.041,A -85,B 0,C 180,E1 11581.595,E2 11581.595} C_VEL
LIN {X 0,Y 539.252,Z 741.018,A -85,B 0,C 180,E1 11583.869,E2 11583.869} C_VEL
LIN {X 0,Y 535.407,Z 774.704,A -85,B 0,C 180,E1 11586.772,E2 11586.772} C_VEL
LIN {X 0,Y 531.811,Z 804.125,A -85,B 0,C 180,E1 11590.211,E2 11590.211} C_VEL
LIN {X 0,Y 529.214,Z 827.144,A -85,B 0,C 180,E1 11593.818,E2 11593.818} C_VEL
LIN {X 0,Y 527.463,Z 845.47,A -85,B 0,C 180,E1 11597.743,E2 11597.743} C_VEL
LIN {X 0,Y 526.453,Z 858.237,A -85,B 0,C 180,E1 11601.721,E2 11601.721} C_VEL
LIN {X 0,Y 526.003,Z 866.05,A -85,B 0,C 180,E1 11605.866,E2 11605.866} C_VEL
LIN {X 0,Y 525.995,Z 868.577,A -85,B 0,C 180,E1 11609.995,E2 11609.995} C_VEL
LIN {X 0,Y 526.042,Z 865.935,A -85,B 0,C 180,E1 11614.125,E2 11614.125} C_VEL
LIN {X 0,Y 526.538,Z 858.002,A -85,B 0,C 180,E1 11618.268,E2 11618.268} C_VEL
LIN {X 0,Y 527.583,Z 844.036,A -85,B 0,C 180,E1 11622.518,E2 11622.518} C_VEL
LIN {X 0,Y 529.412,Z 824.808,A -85,B 0,C 180,E1 11626.512,E2 11626.512} C_VEL
LIN {X 0,Y 532.224,Z 800.662,A -85,B 0,C 180,E1 11630.167,E2 11630.167} C_VEL
LIN {X 0,Y 535.736,Z 771.637,A -85,B 0,C 180,E1 11633.431,E2 11633.431} C_VEL
LIN {X 0,Y 539.446,Z 738.939,A -85,B 0,C 180,E1 11636.191,E2 11636.191} C_VEL
LIN {X 0,Y 543.057,Z 701.952,A -85,B 0,C 180,E1 11638.476,E2 11638.476} C_VEL
LIN {X 0,Y 545.476,Z 662.069,A -85,B 0,C 180,E1 11640.185,E2 11640.185} C_VEL
LIN {X 0,Y 537.361,Z 633.931,A -85,B 0,C 180,E1 11641.585,E2 11641.585} C_VEL
LIN {X 0,Y 523.919,Z 601.31,A -85,B 0,C 180,E1 11643.421,E2 11643.421} C_VEL
LIN {X 0,Y 523.784,Z 601.31,A -85,B 0,C 180,E1 11649.519,E2 11649.519} C_VEL
LIN {X 0,Y 523.832,Z 601.31,A -85,B 0,C 180,E1 11653.958,E2 11653.958} C_VEL
LIN {X 0,Y 523.74,Z 601.31,A -85,B 0,C 180,E1 11660.484,E2 11660.484} C_VEL
LIN {X 0,Y 523.904,Z 601.31,A -85,B 0,C 180,E1 11666.997,E2 11666.997} C_VEL
LIN {X 0,Y 524.058,Z 601.31,A -85,B 0,C 180,E1 11672.453,E2 11672.453} C_VEL
LIN {X 0,Y 524.184,Z 601.31,A -85,B 0,C 180,E1 11674.945,E2 11674.945} C_VEL
LIN {X 0,Y 539.307,Z 650.135,A -85,B 0,C 180,E1 11676.556,E2 11676.556} C_VEL
LIN {X 0,Y 537.743,Z 699.034,A -85,B 0,C 180,E1 11677.521,E2 11677.521} C_VEL
LIN {X 0,Y 535.756,Z 736.62,A -85,B 0,C 180,E1 11678.912,E2 11678.912} C_VEL
LIN {X 0,Y 533.385,Z 770.53,A -85,B 0,C 180,E1 11680.831,E2 11680.831} C_VEL
LIN {X 0,Y 531.196,Z 800.581,A -85,B 0,C 180,E1 11683.24,E2 11683.24} C_VEL
LIN {X 0,Y 529.265,Z 826.776,A -85,B 0,C 180,E1 11686.133,E2 11686.133} C_VEL
LIN {X 0,Y 527.765,Z 848.36,A -85,B 0,C 180,E1 11689.458,E2 11689.458} C_VEL
LIN {X 0,Y 526.996,Z 863.624,A -85,B 0,C 180,E1 11692.88,E2 11692.88} C_VEL
LIN {X 0,Y 526.677,Z 872.208,A -85,B 0,C 180,E1 11695.879,E2 11695.879} C_VEL
LIN {X 0,Y 526.639,Z 876.247,A -85,B 0,C 180,E1 11698.354,E2 11698.354} C_VEL
LIN {X 0,Y 526.716,Z 877.565,A -85,B 0,C 180,E1 11701.65,E2 11701.65} C_VEL
LIN {X 0,Y 527.303,Z 874.08,A -85,B 0,C 180,E1 11704.946,E2 11704.946} C_VEL
LIN {X 0,Y 528.29,Z 864.776,A -85,B 0,C 180,E1 11708.488,E2 11708.488} C_VEL
LIN {X 0,Y 529.783,Z 850.216,A -85,B 0,C 180,E1 11711.758,E2 11711.758} C_VEL
LIN {X 0,Y 531.634,Z 830.008,A -85,B 0,C 180,E1 11714.862,E2 11714.862} C_VEL
LIN {X 0,Y 534.167,Z 804.373,A -85,B 0,C 180,E1 11717.646,E2 11717.646} C_VEL
LIN {X 0,Y 537,Z 772.927,A -85,B 0,C 180,E1 11720.111,E2 11720.111} C_VEL
LIN {X 0,Y 540.03,Z 735.788,A -85,B 0,C 180,E1 11722.167,E2 11722.167} C_VEL
LIN {X 0,Y 543.144,Z 694.015,A -85,B 0,C 180,E1 11723.697,E2 11723.697} C_VEL
LIN {X 0,Y 545.308,Z 650.845,A -85,B 0,C 180,E1 11724.773,E2 11724.773} C_VEL
LIN {X 0,Y 534.958,Z 623.892,A -85,B 0,C 180,E1 11726.487,E2 11726.487} C_VEL
LIN {X 0,Y 525.075,Z 605.164,A -85,B 0,C 180,E1 11728.232,E2 11728.232} C_VEL
LIN {X 0,Y 524.042,Z 601.31,A -85,B 0,C 180,E1 11728.609,E2 11728.609} C_VEL
LIN {X 0,Y 523.929,Z 601.31,A -85,B 0,C 180,E1 11733.326,E2 11733.326} C_VEL
LIN {X 0,Y 523.812,Z 601.31,A -85,B 0,C 180,E1 11739.515,E2 11739.515} C_VEL
LIN {X 0,Y 523.826,Z 601.31,A -85,B 0,C 180,E1 11743.956,E2 11743.956} C_VEL
LIN {X 0,Y 523.799,Z 601.31,A -85,B 0,C 180,E1 11746.445,E2 11746.445} C_VEL
LIN {X 0,Y 526.216,Z 606.961,A -85,B 0,C 180,E1 11746.898,E2 11746.898} C_VEL
LIN {X 0,Y 538.388,Z 629.732,A -85,B 0,C 180,E1 11748.697,E2 11748.697} C_VEL
LIN {X 0,Y 548.18,Z 655.464,A -85,B 0,C 180,E1 11750.016,E2 11750.016} C_VEL
LIN {X 0,Y 555.515,Z 679.197,A -85,B 0,C 180,E1 11750.962,E2 11750.962} C_VEL
LIN {X 0,Y 553.146,Z 726.973,A -85,B 0,C 180,E1 11751.968,E2 11751.968} C_VEL
LIN {X 0,Y 549.414,Z 771.914,A -85,B 0,C 180,E1 11753.565,E2 11753.565} C_VEL
LIN {X 0,Y 546.632,Z 800.872,A -85,B 0,C 180,E1 11754.989,E2 11754.989} C_VEL
LIN {X 0,Y 541.356,Z 816.215,A -85,B 0,C 180,E1 11755.693,E2 11755.693} C_VEL
LIN {X 0,Y 535.867,Z 831.125,A -85,B 0,C 180,E1 11756.48,E2 11756.48} C_VEL
LIN {X 0,Y 530.84,Z 869.793,A -85,B 0,C 180,E1 11759.564,E2 11759.564} C_VEL
LIN {X 0,Y 526.238,Z 905.175,A -85,B 0,C 180,E1 11763.255,E2 11763.255} C_VEL
LIN {X 0,Y 522.503,Z 935.751,A -85,B 0,C 180,E1 11767.409,E2 11767.409} C_VEL
LIN {X 0,Y 519.76,Z 961.147,A -85,B 0,C 180,E1 11771.961,E2 11771.961} C_VEL
LIN {X 0,Y 518.286,Z 979.677,A -85,B 0,C 180,E1 11776.479,E2 11776.479} C_VEL
LIN {X 0,Y 517.729,Z 992.023,A -85,B 0,C 180,E1 11780.742,E2 11780.742} C_VEL
LIN {X 0,Y 517.56,Z 999.528,A -85,B 0,C 180,E1 11784.966,E2 11784.966} C_VEL
LIN {X 0,Y 517.541,Z 1002.412,A -85,B 0,C 180,E1 11788.327,E2 11788.327} C_VEL
LIN {X 0,Y 517.429,Z 1002.503,A -85,B 0,C 180,E1 11791.683,E2 11791.683} C_VEL
LIN {X 0,Y 517.521,Z 999.218,A -85,B 0,C 180,E1 11795.569,E2 11795.569} C_VEL
LIN {X 0,Y 517.746,Z 990.612,A -85,B 0,C 180,E1 11800.118,E2 11800.118} C_VEL
LIN {X 0,Y 518.48,Z 977.948,A -85,B 0,C 180,E1 11804.388,E2 11804.388} C_VEL
LIN {X 0,Y 520.189,Z 958.237,A -85,B 0,C 180,E1 11809.049,E2 11809.049} C_VEL
LIN {X 0,Y 523.13,Z 934.511,A -85,B 0,C 180,E1 11813.248,E2 11813.248} C_VEL
LIN {X 0,Y 527.236,Z 905.275,A -85,B 0,C 180,E1 11817.244,E2 11817.244} C_VEL
LIN {X 0,Y 532.279,Z 870.241,A -85,B 0,C 180,E1 11820.926,E2 11820.926} C_VEL
LIN {X 0,Y 537.746,Z 831.774,A -85,B 0,C 180,E1 11824.006,E2 11824.006} C_VEL
LIN {X 0,Y 543.313,Z 787.897,A -85,B 0,C 180,E1 11826.597,E2 11826.597} C_VEL
LIN {X 0,Y 547.855,Z 743.35,A -85,B 0,C 180,E1 11828.446,E2 11828.446} C_VEL
LIN {X 0,Y 550.909,Z 697.732,A -85,B 0,C 180,E1 11829.648,E2 11829.648} C_VEL
LIN {X 0,Y 551.072,Z 679.398,A -85,B 0,C 180,E1 11829.999,E2 11829.999} C_VEL
LIN {X 0,Y 515.934,Z 601.31,A -85,B 0,C 180,E1 11833.765,E2 11833.765} C_VEL
LIN {X 0,Y 515.806,Z 601.31,A -85,B 0,C 180,E1 11839.804,E2 11839.804} C_VEL
LIN {X 0,Y 515.858,Z 601.31,A -85,B 0,C 180,E1 11846.083,E2 11846.083} C_VEL
LIN {X 0,Y 516.088,Z 601.31,A -85,B 0,C 180,E1 11851.986,E2 11851.986} C_VEL
LIN {X 0,Y 516.288,Z 601.31,A -85,B 0,C 180,E1 11857.575,E2 11857.575} C_VEL
LIN {X 0,Y 516.431,Z 601.31,A -85,B 0,C 180,E1 11862.94,E2 11862.94} C_VEL
LIN {X 0,Y 516.581,Z 601.31,A -85,B 0,C 180,E1 11868.152,E2 11868.152} C_VEL
LIN {X 0,Y 516.869,Z 601.31,A -85,B 0,C 180,E1 11873.265,E2 11873.265} C_VEL
LIN {X 0,Y 517.018,Z 601.31,A -85,B 0,C 180,E1 11878.319,E2 11878.319} C_VEL
LIN {X 0,Y 517.004,Z 601.31,A -85,B 0,C 180,E1 11883.357,E2 11883.357} C_VEL
LIN {X 0,Y 516.746,Z 601.31,A -85,B 0,C 180,E1 11888.427,E2 11888.427} C_VEL
LIN {X 0,Y 516.531,Z 601.31,A -85,B 0,C 180,E1 11894.509,E2 11894.509} C_VEL
LIN {X 0,Y 516.362,Z 601.31,A -85,B 0,C 180,E1 11900.611,E2 11900.611} C_VEL
LIN {X 0,Y 516.146,Z 601.31,A -85,B 0,C 180,E1 11906.117,E2 11906.117} C_VEL
LIN {X 0,Y 515.992,Z 601.31,A -85,B 0,C 180,E1 11911.899,E2 11911.899} C_VEL
LIN {X 0,Y 515.866,Z 601.31,A -85,B 0,C 180,E1 11918.072,E2 11918.072} C_VEL
LIN {X 0,Y 515.841,Z 601.31,A -85,B 0,C 180,E1 11924.811,E2 11924.811} C_VEL
LIN {X 0,Y 515.796,Z 601.31,A -85,B 0,C 180,E1 11929.781,E2 11929.781} C_VEL
LIN {X 0,Y 516.022,Z 601.991,A -85,B 0,C 180,E1 11935.975,E2 11935.975} C_VEL
LIN {X 0,Y 535.218,Z 649.053,A -85,B 0,C 180,E1 11938.602,E2 11938.602} C_VEL
LIN {X 0,Y 538.903,Z 666.77,A -85,B 0,C 180,E1 11939.475,E2 11939.475} C_VEL
LIN {X 0,Y 535.888,Z 705.794,A -85,B 0,C 180,E1 11941.198,E2 11941.198} C_VEL
LIN {X 0,Y 532.158,Z 742.117,A -85,B 0,C 180,E1 11943.52,E2 11943.52} C_VEL
LIN {X 0,Y 528.262,Z 774.376,A -85,B 0,C 180,E1 11946.319,E2 11946.319} C_VEL
LIN {X 0,Y 524.57,Z 803.539,A -85,B 0,C 180,E1 11949.715,E2 11949.715} C_VEL
LIN {X 0,Y 521.758,Z 826.844,A -85,B 0,C 180,E1 11953.354,E2 11953.354} C_VEL
LIN {X 0,Y 519.818,Z 845.478,A -85,B 0,C 180,E1 11957.324,E2 11957.324} C_VEL
LIN {X 0,Y 518.68,Z 859.197,A -85,B 0,C 180,E1 11961.596,E2 11961.596} C_VEL
LIN {X 0,Y 518.196,Z 867.029,A -85,B 0,C 180,E1 11965.803,E2 11965.803} C_VEL
LIN {X 0,Y 518.174,Z 869.563,A -85,B 0,C 180,E1 11969.995,E2 11969.995} C_VEL
LIN {X 0,Y 518.232,Z 866.914,A -85,B 0,C 180,E1 11974.187,E2 11974.187} C_VEL
LIN {X 0,Y 518.763,Z 858.965,A -85,B 0,C 180,E1 11978.393,E2 11978.393} C_VEL
LIN {X 0,Y 519.897,Z 844.979,A -85,B 0,C 180,E1 11982.707,E2 11982.707} C_VEL
LIN {X 0,Y 521.766,Z 826.331,A -85,B 0,C 180,E1 11986.649,E2 11986.649} C_VEL
LIN {X 0,Y 524.86,Z 801.365,A -85,B 0,C 180,E1 11990.485,E2 11990.485} C_VEL
LIN {X 0,Y 528.619,Z 771.392,A -85,B 0,C 180,E1 11993.878,E2 11993.878} C_VEL
LIN {X 0,Y 532.58,Z 738.132,A -85,B 0,C 180,E1 11996.685,E2 11996.685} C_VEL
LIN {X 0,Y 536.199,Z 701.863,A -85,B 0,C 180,E1 11998.913,E2 11998.913} C_VEL
LIN {X 0,Y 538.39,Z 663.328,A -85,B 0,C 180,E1 12000.593,E2 12000.593} C_VEL
LIN {X 0,Y 530.969,Z 637.314,A -85,B 0,C 180,E1 12001.924,E2 12001.924} C_VEL
LIN {X 0,Y 516.041,Z 601.31,A -85,B 0,C 180,E1 12004.003,E2 12004.003} C_VEL
LIN {X 0,Y 515.861,Z 601.31,A -85,B 0,C 180,E1 12010.249,E2 12010.249} C_VEL
LIN {X 0,Y 515.831,Z 601.31,A -85,B 0,C 180,E1 12015.187,E2 12015.187} C_VEL
LIN {X 0,Y 515.828,Z 601.31,A -85,B 0,C 180,E1 12021.925,E2 12021.925} C_VEL
LIN {X 0,Y 516.018,Z 601.31,A -85,B 0,C 180,E1 12028.371,E2 12028.371} C_VEL
LIN {X 0,Y 516.26,Z 601.31,A -85,B 0,C 180,E1 12034.559,E2 12034.559} C_VEL
LIN {X 0,Y 531.91,Z 651.947,A -85,B 0,C 180,E1 12036.271,E2 12036.271} C_VEL
LIN {X 0,Y 530.308,Z 699.741,A -85,B 0,C 180,E1 12037.242,E2 12037.242} C_VEL
LIN {X 0,Y 528.273,Z 736.871,A -85,B 0,C 180,E1 12038.64,E2 12038.64} C_VEL
LIN {X 0,Y 525.764,Z 771.803,A -85,B 0,C 180,E1 12040.652,E2 12040.652} C_VEL
LIN {X 0,Y 523.428,Z 802.649,A -85,B 0,C 180,E1 12043.179,E2 12043.179} C_VEL
LIN {X 0,Y 521.468,Z 828.692,A -85,B 0,C 180,E1 12046.135,E2 12046.135} C_VEL
LIN {X 0,Y 519.907,Z 850.011,A -85,B 0,C 180,E1 12049.509,E2 12049.509} C_VEL
LIN {X 0,Y 519.184,Z 864.567,A -85,B 0,C 180,E1 12052.833,E2 12052.833} C_VEL
LIN {X 0,Y 518.853,Z 873.072,A -85,B 0,C 180,E1 12055.816,E2 12055.816} C_VEL
LIN {X 0,Y 518.817,Z 877.231,A -85,B 0,C 180,E1 12058.329,E2 12058.329} C_VEL
LIN {X 0,Y 518.896,Z 878.669,A -85,B 0,C 180,E1 12061.675,E2 12061.675} C_VEL
LIN {X 0,Y 519.552,Z 875.308,A -85,B 0,C 180,E1 12065.02,E2 12065.02} C_VEL
LIN {X 0,Y 520.491,Z 866.925,A -85,B 0,C 180,E1 12068.37,E2 12068.37} C_VEL
LIN {X 0,Y 522.035,Z 852.773,A -85,B 0,C 180,E1 12071.722,E2 12071.722} C_VEL
LIN {X 0,Y 524.075,Z 833.043,A -85,B 0,C 180,E1 12074.88,E2 12074.88} C_VEL
LIN {X 0,Y 526.788,Z 807.236,A -85,B 0,C 180,E1 12077.793,E2 12077.793} C_VEL
LIN {X 0,Y 529.666,Z 776.714,A -85,B 0,C 180,E1 12080.293,E2 12080.293} C_VEL
LIN {X 0,Y 532.864,Z 740.488,A -85,B 0,C 180,E1 12082.401,E2 12082.401} C_VEL
LIN {X 0,Y 536.339,Z 697.733,A -85,B 0,C 180,E1 12084.068,E2 12084.068} C_VEL
LIN {X 0,Y 538.877,Z 653.204,A -85,B 0,C 180,E1 12085.221,E2 12085.221} C_VEL
LIN {X 0,Y 529.04,Z 627.091,A -85,B 0,C 180,E1 12086.98,E2 12086.98} C_VEL
LIN {X 0,Y 518.581,Z 607.017,A -85,B 0,C 180,E1 12088.999,E2 12088.999} C_VEL
LIN {X 0,Y 516.079,Z 601.31,A -85,B 0,C 180,E1 12089.727,E2 12089.727} C_VEL
LIN {X 0,Y 515.944,Z 601.31,A -85,B 0,C 180,E1 12095.963,E2 12095.963} C_VEL
LIN {X 0,Y 515.848,Z 601.31,A -85,B 0,C 180,E1 12102.491,E2 12102.491} C_VEL
LIN {X 0,Y 515.841,Z 601.524,A -85,B 0,C 180,E1 12105.349,E2 12105.349} C_VEL
LIN {X 0,Y 518.39,Z 607.08,A -85,B 0,C 180,E1 12105.891,E2 12105.891} C_VEL
LIN {X 0,Y 529.57,Z 626.699,A -85,B 0,C 180,E1 12107.75,E2 12107.75} C_VEL
LIN {X 0,Y 539.926,Z 651.325,A -85,B 0,C 180,E1 12109.251,E2 12109.251} C_VEL
LIN {X 0,Y 548.947,Z 682.471,A -85,B 0,C 180,E1 12110.542,E2 12110.542} C_VEL
LIN {X 0,Y 546.403,Z 728.585,A -85,B 0,C 180,E1 12111.567,E2 12111.567} C_VEL
LIN {X 0,Y 542.598,Z 771.789,A -85,B 0,C 180,E1 12113.142,E2 12113.142} C_VEL
LIN {X 0,Y 537.892,Z 815.498,A -85,B 0,C 180,E1 12115.456,E2 12115.456} C_VEL
LIN {X 0,Y 535.867,Z 831.125,A -85,B 0,C 180,E1 12116.48,E2 12116.48} C_VEL
LIN {X 0,Y 530.417,Z 845.672,A -85,B 0,C 180,E1 12117.371,E2 12117.371} C_VEL
LIN {X 0,Y 524.944,Z 859.637,A -85,B 0,C 180,E1 12118.346,E2 12118.346} C_VEL
LIN {X 0,Y 520.094,Z 894.683,A -85,B 0,C 180,E1 12121.8,E2 12121.8} C_VEL
LIN {X 0,Y 515.941,Z 925.653,A -85,B 0,C 180,E1 12125.728,E2 12125.728} C_VEL
LIN {X 0,Y 512.705,Z 953.483,A -85,B 0,C 180,E1 12130.361,E2 12130.361} C_VEL
LIN {X 0,Y 510.832,Z 973.931,A -85,B 0,C 180,E1 12134.962,E2 12134.962} C_VEL
LIN {X 0,Y 510.014,Z 987.399,A -85,B 0,C 180,E1 12139.131,E2 12139.131} C_VEL
LIN {X 0,Y 509.726,Z 996.114,A -85,B 0,C 180,E1 12143.176,E2 12143.176} C_VEL
LIN {X 0,Y 509.624,Z 1000.422,A -85,B 0,C 180,E1 12146.596,E2 12146.596} C_VEL
LIN {X 0,Y 509.69,Z 1001.968,A -85,B 0,C 180,E1 12150.005,E2 12150.005} C_VEL
LIN {X 0,Y 509.703,Z 998.987,A -85,B 0,C 180,E1 12155.121,E2 12155.121} C_VEL
LIN {X 0,Y 509.827,Z 990.75,A -85,B 0,C 180,E1 12159.844,E2 12159.844} C_VEL
LIN {X 0,Y 510.687,Z 977.005,A -85,B 0,C 180,E1 12164.612,E2 12164.612} C_VEL
LIN {X 0,Y 512.514,Z 956.784,A -85,B 0,C 180,E1 12169.431,E2 12169.431} C_VEL
LIN {X 0,Y 515.76,Z 931.887,A -85,B 0,C 180,E1 12173.83,E2 12173.83} C_VEL
